P[2666]{
   GP1:
	UF : 0, UT : 6,		CONFIG : 'N U T, 0, 0, 0',
	X =  -88.796  mm,	Y =   -332.200  mm,	Z =   -251.035  mm,
	W =  90.000 deg,	P =   0.000 deg,	R =   90.000 deg
};
P[2667]{
   GP1:
	UF : 0, UT : 6,		CONFIG : 'N U T, 0, 0, 0',
	X =  -94.111  mm,	Y =   -335.387  mm,	Z =   -251.321  mm,
	W =  90.000 deg,	P =   0.000 deg,	R =   90.000 deg
};
P[2668]{
   GP1:
	UF : 0, UT : 6,		CONFIG : 'N U T, 0, 0, 0',
	X =  -94.874  mm,	Y =   -335.891  mm,	Z =   -251.475  mm,
	W =  90.000 deg,	P =   0.000 deg,	R =   90.000 deg
};
P[2669]{
   GP1:
	UF : 0, UT : 6,		CONFIG : 'N U T, 0, 0, 0',
	X =  -96.510  mm,	Y =   -336.847  mm,	Z =   -251.505  mm,
	W =  90.000 deg,	P =   0.000 deg,	R =   90.000 deg
};
P[2670]{
   GP1:
	UF : 0, UT : 6,		CONFIG : 'N U T, 0, 0, 0',
	X =  -98.758  mm,	Y =   -337.951  mm,	Z =   -251.032  mm,
	W =  90.000 deg,	P =   0.000 deg,	R =   90.000 deg
};
P[2671]{
   GP1:
	UF : 0, UT : 6,		CONFIG : 'N U T, 0, 0, 0',
	X =  -100.678  mm,	Y =   -339.223  mm,	Z =   -251.429  mm,
	W =  90.000 deg,	P =   0.000 deg,	R =   90.000 deg
};
P[2672]{
   GP1:
	UF : 0, UT : 6,		CONFIG : 'N U T, 0, 0, 0',
	X =  -102.192  mm,	Y =   -340.019  mm,	Z =   -251.240  mm,
	W =  90.000 deg,	P =   0.000 deg,	R =   90.000 deg
};
P[2673]{
   GP1:
	UF : 0, UT : 6,		CONFIG : 'N U T, 0, 0, 0',
	X =  -103.313  mm,	Y =   -340.755  mm,	Z =   -251.454  mm,
	W =  90.000 deg,	P =   0.000 deg,	R =   90.000 deg
};
P[2674]{
   GP1:
	UF : 0, UT : 6,		CONFIG : 'N U T, 0, 0, 0',
	X =  -105.295  mm,	Y =   -341.722  mm,	Z =   -251.025  mm,
	W =  90.000 deg,	P =   0.000 deg,	R =   90.000 deg
};
P[2675]{
   GP1:
	UF : 0, UT : 6,		CONFIG : 'N U T, 0, 0, 0',
	X =  -106.428  mm,	Y =   -342.386  mm,	Z =   -251.049  mm,
	W =  90.000 deg,	P =   0.000 deg,	R =   90.000 deg
};
P[2676]{
   GP1:
	UF : 0, UT : 6,		CONFIG : 'N U T, 0, 0, 0',
	X =  -108.033  mm,	Y =   -343.483  mm,	Z =   -251.461  mm,
	W =  90.000 deg,	P =   0.000 deg,	R =   90.000 deg
};
P[2677]{
   GP1:
	UF : 0, UT : 6,		CONFIG : 'N U T, 0, 0, 0',
	X =  -108.863  mm,	Y =   -343.861  mm,	Z =   -251.217  mm,
	W =  90.000 deg,	P =   0.000 deg,	R =   90.000 deg
};
P[2678]{
   GP1:
	UF : 0, UT : 6,		CONFIG : 'N U T, 0, 0, 0',
	X =  -110.601  mm,	Y =   -344.960  mm,	Z =   -251.448  mm,
	W =  90.000 deg,	P =   0.000 deg,	R =   90.000 deg
};
P[2679]{
   GP1:
	UF : 0, UT : 6,		CONFIG : 'N U T, 0, 0, 0',
	X =  -113.227  mm,	Y =   -346.434  mm,	Z =   -251.345  mm,
	W =  90.000 deg,	P =   0.000 deg,	R =   90.000 deg
};
P[2680]{
   GP1:
	UF : 0, UT : 6,		CONFIG : 'N U T, 0, 0, 0',
	X =  -116.933  mm,	Y =   -348.507  mm,	Z =   -251.183  mm,
	W =  90.000 deg,	P =   0.000 deg,	R =   90.000 deg
};
P[2681]{
   GP1:
	UF : 0, UT : 6,		CONFIG : 'N U T, 0, 0, 0',
	X =  -119.089  mm,	Y =   -350.044  mm,	Z =   -251.339  mm,
	W =  90.000 deg,	P =   0.000 deg,	R =   90.000 deg
};
P[2682]{
   GP1:
	UF : 0, UT : 6,		CONFIG : 'N U T, 0, 0, 0',
	X =  -121.292  mm,	Y =   -352.219  mm,	Z =   -251.419  mm,
	W =  90.000 deg,	P =   0.000 deg,	R =   90.000 deg
};
P[2683]{
   GP1:
	UF : 0, UT : 6,		CONFIG : 'N U T, 0, 0, 0',
	X =  -122.707  mm,	Y =   -354.283  mm,	Z =   -251.379  mm,
	W =  90.000 deg,	P =   0.000 deg,	R =   90.000 deg
};
P[2684]{
   GP1:
	UF : 0, UT : 6,		CONFIG : 'N U T, 0, 0, 0',
	X =  -123.543  mm,	Y =   -356.394  mm,	Z =   -251.512  mm,
	W =  90.000 deg,	P =   0.000 deg,	R =   90.000 deg
};
P[2685]{
   GP1:
	UF : 0, UT : 6,		CONFIG : 'N U T, 0, 0, 0',
	X =  -123.974  mm,	Y =   -357.288  mm,	Z =   -251.247  mm,
	W =  90.000 deg,	P =   0.000 deg,	R =   90.000 deg
};
P[2686]{
   GP1:
	UF : 0, UT : 6,		CONFIG : 'N U T, 0, 0, 0',
	X =  -124.171  mm,	Y =   -358.080  mm,	Z =   -251.154  mm,
	W =  90.000 deg,	P =   0.000 deg,	R =   90.000 deg
};
P[2687]{
   GP1:
	UF : 0, UT : 6,		CONFIG : 'N U T, 0, 0, 0',
	X =  -124.217  mm,	Y =   -359.462  mm,	Z =   -251.503  mm,
	W =  90.000 deg,	P =   0.000 deg,	R =   90.000 deg
};
P[2688]{
   GP1:
	UF : 0, UT : 6,		CONFIG : 'N U T, 0, 0, 0',
	X =  -124.347  mm,	Y =   -360.646  mm,	Z =   -251.277  mm,
	W =  90.000 deg,	P =   0.000 deg,	R =   90.000 deg
};
P[2689]{
   GP1:
	UF : 0, UT : 6,		CONFIG : 'N U T, 0, 0, 0',
	X =  -124.228  mm,	Y =   -361.334  mm,	Z =   -251.466  mm,
	W =  90.000 deg,	P =   0.000 deg,	R =   90.000 deg
};
P[2690]{
   GP1:
	UF : 0, UT : 6,		CONFIG : 'N U T, 0, 0, 0',
	X =  -124.026  mm,	Y =   -363.050  mm,	Z =   -251.504  mm,
	W =  90.000 deg,	P =   0.000 deg,	R =   90.000 deg
};
P[2691]{
   GP1:
	UF : 0, UT : 6,		CONFIG : 'N U T, 0, 0, 0',
	X =  -123.894  mm,	Y =   -364.249  mm,	Z =   -251.149  mm,
	W =  90.000 deg,	P =   0.000 deg,	R =   90.000 deg
};
P[2692]{
   GP1:
	UF : 0, UT : 6,		CONFIG : 'N U T, 0, 0, 0',
	X =  -123.534  mm,	Y =   -365.086  mm,	Z =   -251.490  mm,
	W =  90.000 deg,	P =   0.000 deg,	R =   90.000 deg
};
P[2693]{
   GP1:
	UF : 0, UT : 6,		CONFIG : 'N U T, 0, 0, 0',
	X =  -123.293  mm,	Y =   -365.993  mm,	Z =   -251.111  mm,
	W =  90.000 deg,	P =   0.000 deg,	R =   90.000 deg
};
P[2694]{
   GP1:
	UF : 0, UT : 6,		CONFIG : 'N U T, 0, 0, 0',
	X =  -117.435  mm,	Y =   -376.328  mm,	Z =   -251.323  mm,
	W =  90.000 deg,	P =   0.000 deg,	R =   90.000 deg
};
P[2695]{
   GP1:
	UF : 0, UT : 6,		CONFIG : 'N U T, 0, 0, 0',
	X =  -116.602  mm,	Y =   -377.647  mm,	Z =   -251.497  mm,
	W =  90.000 deg,	P =   0.000 deg,	R =   90.000 deg
};
P[2696]{
   GP1:
	UF : 0, UT : 6,		CONFIG : 'N U T, 0, 0, 0',
	X =  -116.076  mm,	Y =   -378.576  mm,	Z =   -251.473  mm,
	W =  90.000 deg,	P =   0.000 deg,	R =   90.000 deg
};
P[2697]{
   GP1:
	UF : 0, UT : 6,		CONFIG : 'N U T, 0, 0, 0',
	X =  -115.720  mm,	Y =   -379.277  mm,	Z =   -251.355  mm,
	W =  90.000 deg,	P =   0.000 deg,	R =   90.000 deg
};
P[2698]{
   GP1:
	UF : 0, UT : 6,		CONFIG : 'N U T, 0, 0, 0',
	X =  -114.684  mm,	Y =   -380.969  mm,	Z =   -251.496  mm,
	W =  90.000 deg,	P =   0.000 deg,	R =   90.000 deg
};
P[2699]{
   GP1:
	UF : 0, UT : 6,		CONFIG : 'N U T, 0, 0, 0',
	X =  -113.664  mm,	Y =   -382.827  mm,	Z =   -251.369  mm,
	W =  90.000 deg,	P =   0.000 deg,	R =   90.000 deg
};
P[2700]{
   GP1:
	UF : 0, UT : 6,		CONFIG : 'N U T, 0, 0, 0',
	X =  -112.347  mm,	Y =   -385.040  mm,	Z =   -251.463  mm,
	W =  90.000 deg,	P =   0.000 deg,	R =   90.000 deg
};
P[2701]{
   GP1:
	UF : 0, UT : 6,		CONFIG : 'N U T, 0, 0, 0',
	X =  -111.510  mm,	Y =   -386.475  mm,	Z =   -251.485  mm,
	W =  90.000 deg,	P =   0.000 deg,	R =   90.000 deg
};
P[2702]{
   GP1:
	UF : 0, UT : 6,		CONFIG : 'N U T, 0, 0, 0',
	X =  -110.653  mm,	Y =   -388.090  mm,	Z =   -251.300  mm,
	W =  90.000 deg,	P =   0.000 deg,	R =   90.000 deg
};
P[2703]{
   GP1:
	UF : 0, UT : 6,		CONFIG : 'N U T, 0, 0, 0',
	X =  -109.246  mm,	Y =   -390.539  mm,	Z =   -251.286  mm,
	W =  90.000 deg,	P =   0.000 deg,	R =   90.000 deg
};
P[2704]{
   GP1:
	UF : 0, UT : 6,		CONFIG : 'N U T, 0, 0, 0',
	X =  -107.328  mm,	Y =   -393.699  mm,	Z =   -251.513  mm,
	W =  90.000 deg,	P =   0.000 deg,	R =   90.000 deg
};
P[2705]{
   GP1:
	UF : 0, UT : 6,		CONFIG : 'N U T, 0, 0, 0',
	X =  -106.006  mm,	Y =   -396.158  mm,	Z =   -251.273  mm,
	W =  90.000 deg,	P =   0.000 deg,	R =   90.000 deg
};
P[2706]{
   GP1:
	UF : 0, UT : 6,		CONFIG : 'N U T, 0, 0, 0',
	X =  -102.398  mm,	Y =   -402.502  mm,	Z =   -251.140  mm,
	W =  90.000 deg,	P =   0.000 deg,	R =   90.000 deg
};
P[2707]{
   GP1:
	UF : 0, UT : 6,		CONFIG : 'N U T, 0, 0, 0',
	X =  -101.351  mm,	Y =   -404.270  mm,	Z =   -251.205  mm,
	W =  90.000 deg,	P =   0.000 deg,	R =   90.000 deg
};
P[2708]{
   GP1:
	UF : 0, UT : 6,		CONFIG : 'N U T, 0, 0, 0',
	X =  -100.892  mm,	Y =   -404.878  mm,	Z =   -251.465  mm,
	W =  90.000 deg,	P =   0.000 deg,	R =   90.000 deg
};
P[2709]{
   GP1:
	UF : 0, UT : 6,		CONFIG : 'N U T, 0, 0, 0',
	X =  -97.701  mm,	Y =   -410.426  mm,	Z =   -251.435  mm,
	W =  90.000 deg,	P =   0.000 deg,	R =   90.000 deg
};
P[2710]{
   GP1:
	UF : 0, UT : 6,		CONFIG : 'N U T, 0, 0, 0',
	X =  -96.296  mm,	Y =   -413.012  mm,	Z =   -251.222  mm,
	W =  90.000 deg,	P =   0.000 deg,	R =   90.000 deg
};
P[2711]{
   GP1:
	UF : 0, UT : 6,		CONFIG : 'N U T, 0, 0, 0',
	X =  -95.621  mm,	Y =   -413.979  mm,	Z =   -251.505  mm,
	W =  90.000 deg,	P =   0.000 deg,	R =   90.000 deg
};
P[2712]{
   GP1:
	UF : 0, UT : 6,		CONFIG : 'N U T, 0, 0, 0',
	X =  -94.896  mm,	Y =   -415.279  mm,	Z =   -251.445  mm,
	W =  90.000 deg,	P =   0.000 deg,	R =   90.000 deg
};
P[2713]{
   GP1:
	UF : 0, UT : 6,		CONFIG : 'N U T, 0, 0, 0',
	X =  -94.523  mm,	Y =   -416.116  mm,	Z =   -251.175  mm,
	W =  90.000 deg,	P =   0.000 deg,	R =   90.000 deg
};
P[2714]{
   GP1:
	UF : 0, UT : 6,		CONFIG : 'N U T, 0, 0, 0',
	X =  -94.072  mm,	Y =   -416.738  mm,	Z =   -251.398  mm,
	W =  90.000 deg,	P =   0.000 deg,	R =   90.000 deg
};
P[2715]{
   GP1:
	UF : 0, UT : 6,		CONFIG : 'N U T, 0, 0, 0',
	X =  -93.224  mm,	Y =   -418.286  mm,	Z =   -251.287  mm,
	W =  90.000 deg,	P =   0.000 deg,	R =   90.000 deg
};
P[2716]{
   GP1:
	UF : 0, UT : 6,		CONFIG : 'N U T, 0, 0, 0',
	X =  -92.392  mm,	Y =   -419.819  mm,	Z =   -251.157  mm,
	W =  90.000 deg,	P =   0.000 deg,	R =   90.000 deg
};
P[2717]{
   GP1:
	UF : 0, UT : 6,		CONFIG : 'N U T, 0, 0, 0',
	X =  -89.616  mm,	Y =   -424.487  mm,	Z =   -251.353  mm,
	W =  90.000 deg,	P =   0.000 deg,	R =   90.000 deg
};
P[2718]{
   GP1:
	UF : 0, UT : 6,		CONFIG : 'N U T, 0, 0, 0',
	X =  -88.935  mm,	Y =   -425.905  mm,	Z =   -251.019  mm,
	W =  90.000 deg,	P =   0.000 deg,	R =   90.000 deg
};
P[2719]{
   GP1:
	UF : 0, UT : 6,		CONFIG : 'N U T, 0, 0, 0',
	X =  -88.296  mm,	Y =   -426.877  mm,	Z =   -251.210  mm,
	W =  90.000 deg,	P =   0.000 deg,	R =   90.000 deg
};
P[2720]{
   GP1:
	UF : 0, UT : 6,		CONFIG : 'N U T, 0, 0, 0',
	X =  -87.498  mm,	Y =   -428.081  mm,	Z =   -251.458  mm,
	W =  90.000 deg,	P =   0.000 deg,	R =   90.000 deg
};
P[2721]{
   GP1:
	UF : 0, UT : 6,		CONFIG : 'N U T, 0, 0, 0',
	X =  -87.062  mm,	Y =   -428.796  mm,	Z =   -251.514  mm,
	W =  90.000 deg,	P =   0.000 deg,	R =   90.000 deg
};
P[2722]{
   GP1:
	UF : 0, UT : 6,		CONFIG : 'N U T, 0, 0, 0',
	X =  -83.860  mm,	Y =   -434.387  mm,	Z =   -251.452  mm,
	W =  90.000 deg,	P =   0.000 deg,	R =   90.000 deg
};
P[2723]{
   GP1:
	UF : 0, UT : 6,		CONFIG : 'N U T, 0, 0, 0',
	X =  -82.430  mm,	Y =   -437.003  mm,	Z =   -251.256  mm,
	W =  90.000 deg,	P =   0.000 deg,	R =   90.000 deg
};
P[2724]{
   GP1:
	UF : 0, UT : 6,		CONFIG : 'N U T, 0, 0, 0',
	X =  -80.657  mm,	Y =   -439.990  mm,	Z =   -251.371  mm,
	W =  90.000 deg,	P =   0.000 deg,	R =   90.000 deg
};
P[2725]{
   GP1:
	UF : 0, UT : 6,		CONFIG : 'N U T, 0, 0, 0',
	X =  -80.143  mm,	Y =   -440.820  mm,	Z =   -251.456  mm,
	W =  90.000 deg,	P =   0.000 deg,	R =   90.000 deg
};
P[2726]{
   GP1:
	UF : 0, UT : 6,		CONFIG : 'N U T, 0, 0, 0',
	X =  -79.054  mm,	Y =   -442.851  mm,	Z =   -251.254  mm,
	W =  90.000 deg,	P =   0.000 deg,	R =   90.000 deg
};
P[2727]{
   GP1:
	UF : 0, UT : 6,		CONFIG : 'N U T, 0, 0, 0',
	X =  -77.555  mm,	Y =   -445.264  mm,	Z =   -251.509  mm,
	W =  90.000 deg,	P =   0.000 deg,	R =   90.000 deg
};
P[2728]{
   GP1:
	UF : 0, UT : 6,		CONFIG : 'N U T, 0, 0, 0',
	X =  -75.494  mm,	Y =   -449.012  mm,	Z =   -251.260  mm,
	W =  90.000 deg,	P =   0.000 deg,	R =   90.000 deg
};
P[2729]{
   GP1:
	UF : 0, UT : 6,		CONFIG : 'N U T, 0, 0, 0',
	X =  -74.771  mm,	Y =   -450.179  mm,	Z =   -251.380  mm,
	W =  90.000 deg,	P =   0.000 deg,	R =   90.000 deg
};
P[2730]{
   GP1:
	UF : 0, UT : 6,		CONFIG : 'N U T, 0, 0, 0',
	X =  -73.079  mm,	Y =   -453.059  mm,	Z =   -251.451  mm,
	W =  90.000 deg,	P =   0.000 deg,	R =   90.000 deg
};
P[2731]{
   GP1:
	UF : 0, UT : 6,		CONFIG : 'N U T, 0, 0, 0',
	X =  -68.696  mm,	Y =   -460.609  mm,	Z =   -251.506  mm,
	W =  90.000 deg,	P =   0.000 deg,	R =   90.000 deg
};
P[2732]{
   GP1:
	UF : 0, UT : 6,		CONFIG : 'N U T, 0, 0, 0',
	X =  -68.326  mm,	Y =   -461.356  mm,	Z =   -251.359  mm,
	W =  90.000 deg,	P =   0.000 deg,	R =   90.000 deg
};
P[2733]{
   GP1:
	UF : 0, UT : 6,		CONFIG : 'N U T, 0, 0, 0',
	X =  -67.778  mm,	Y =   -462.396  mm,	Z =   -251.232  mm,
	W =  90.000 deg,	P =   0.000 deg,	R =   90.000 deg
};
P[2734]{
   GP1:
	UF : 0, UT : 6,		CONFIG : 'N U T, 0, 0, 0',
	X =  -67.192  mm,	Y =   -463.250  mm,	Z =   -251.458  mm,
	W =  90.000 deg,	P =   0.000 deg,	R =   90.000 deg
};
P[2735]{
   GP1:
	UF : 0, UT : 6,		CONFIG : 'N U T, 0, 0, 0',
	X =  -64.146  mm,	Y =   -468.762  mm,	Z =   -251.125  mm,
	W =  90.000 deg,	P =   0.000 deg,	R =   90.000 deg
};
P[2736]{
   GP1:
	UF : 0, UT : 6,		CONFIG : 'N U T, 0, 0, 0',
	X =  -62.301  mm,	Y =   -471.708  mm,	Z =   -251.474  mm,
	W =  90.000 deg,	P =   0.000 deg,	R =   90.000 deg
};
P[2737]{
   GP1:
	UF : 0, UT : 6,		CONFIG : 'N U T, 0, 0, 0',
	X =  -60.967  mm,	Y =   -474.301  mm,	Z =   -251.079  mm,
	W =  90.000 deg,	P =   0.000 deg,	R =   90.000 deg
};
P[2738]{
   GP1:
	UF : 0, UT : 6,		CONFIG : 'N U T, 0, 0, 0',
	X =  -59.945  mm,	Y =   -475.996  mm,	Z =   -251.183  mm,
	W =  90.000 deg,	P =   0.000 deg,	R =   90.000 deg
};
P[2739]{
   GP1:
	UF : 0, UT : 6,		CONFIG : 'N U T, 0, 0, 0',
	X =  -56.961  mm,	Y =   -481.089  mm,	Z =   -251.291  mm,
	W =  90.000 deg,	P =   0.000 deg,	R =   90.000 deg
};
P[2740]{
   GP1:
	UF : 0, UT : 6,		CONFIG : 'N U T, 0, 0, 0',
	X =  -55.926  mm,	Y =   -482.733  mm,	Z =   -251.499  mm,
	W =  90.000 deg,	P =   0.000 deg,	R =   90.000 deg
};
P[2741]{
   GP1:
	UF : 0, UT : 6,		CONFIG : 'N U T, 0, 0, 0',
	X =  -55.119  mm,	Y =   -484.466  mm,	Z =   -251.027  mm,
	W =  90.000 deg,	P =   0.000 deg,	R =   90.000 deg
};
P[2742]{
   GP1:
	UF : 0, UT : 6,		CONFIG : 'N U T, 0, 0, 0',
	X =  -52.807  mm,	Y =   -488.183  mm,	Z =   -251.430  mm,
	W =  90.000 deg,	P =   0.000 deg,	R =   90.000 deg
};
P[2743]{
   GP1:
	UF : 0, UT : 6,		CONFIG : 'N U T, 0, 0, 0',
	X =  -52.049  mm,	Y =   -489.711  mm,	Z =   -251.128  mm,
	W =  90.000 deg,	P =   0.000 deg,	R =   90.000 deg
};
P[2744]{
   GP1:
	UF : 0, UT : 6,		CONFIG : 'N U T, 0, 0, 0',
	X =  -48.701  mm,	Y =   -495.270  mm,	Z =   -251.462  mm,
	W =  90.000 deg,	P =   0.000 deg,	R =   90.000 deg
};
P[2745]{
   GP1:
	UF : 0, UT : 6,		CONFIG : 'N U T, 0, 0, 0',
	X =  -48.119  mm,	Y =   -496.321  mm,	Z =   -251.403  mm,
	W =  90.000 deg,	P =   0.000 deg,	R =   90.000 deg
};
P[2746]{
   GP1:
	UF : 0, UT : 6,		CONFIG : 'N U T, 0, 0, 0',
	X =  -46.469  mm,	Y =   -499.194  mm,	Z =   -251.385  mm,
	W =  90.000 deg,	P =   0.000 deg,	R =   90.000 deg
};
P[2747]{
   GP1:
	UF : 0, UT : 6,		CONFIG : 'N U T, 0, 0, 0',
	X =  -46.266  mm,	Y =   -499.788  mm,	Z =   -251.042  mm,
	W =  90.000 deg,	P =   0.000 deg,	R =   90.000 deg
};
P[2748]{
   GP1:
	UF : 0, UT : 6,		CONFIG : 'N U T, 0, 0, 0',
	X =  -45.082  mm,	Y =   -501.624  mm,	Z =   -251.345  mm,
	W =  90.000 deg,	P =   0.000 deg,	R =   90.000 deg
};
P[2749]{
   GP1:
	UF : 0, UT : 6,		CONFIG : 'N U T, 0, 0, 0',
	X =  -44.497  mm,	Y =   -502.677  mm,	Z =   -251.288  mm,
	W =  90.000 deg,	P =   0.000 deg,	R =   90.000 deg
};
P[2750]{
   GP1:
	UF : 0, UT : 6,		CONFIG : 'N U T, 0, 0, 0',
	X =  -44.054  mm,	Y =   -503.435  mm,	Z =   -251.301  mm,
	W =  90.000 deg,	P =   0.000 deg,	R =   90.000 deg
};
P[2751]{
   GP1:
	UF : 0, UT : 6,		CONFIG : 'N U T, 0, 0, 0',
	X =  -41.974  mm,	Y =   -507.109  mm,	Z =   -251.201  mm,
	W =  90.000 deg,	P =   0.000 deg,	R =   90.000 deg
};
P[2752]{
   GP1:
	UF : 0, UT : 6,		CONFIG : 'N U T, 0, 0, 0',
	X =  -41.447  mm,	Y =   -507.963  mm,	Z =   -251.281  mm,
	W =  90.000 deg,	P =   0.000 deg,	R =   90.000 deg
};
P[2753]{
   GP1:
	UF : 0, UT : 6,		CONFIG : 'N U T, 0, 0, 0',
	X =  -40.849  mm,	Y =   -508.939  mm,	Z =   -251.367  mm,
	W =  90.000 deg,	P =   0.000 deg,	R =   90.000 deg
};
P[2754]{
   GP1:
	UF : 0, UT : 6,		CONFIG : 'N U T, 0, 0, 0',
	X =  -39.722  mm,	Y =   -510.925  mm,	Z =   -251.316  mm,
	W =  90.000 deg,	P =   0.000 deg,	R =   90.000 deg
};
P[2755]{
   GP1:
	UF : 0, UT : 6,		CONFIG : 'N U T, 0, 0, 0',
	X =  -38.820  mm,	Y =   -512.403  mm,	Z =   -251.437  mm,
	W =  90.000 deg,	P =   0.000 deg,	R =   90.000 deg
};
P[2756]{
   GP1:
	UF : 0, UT : 6,		CONFIG : 'N U T, 0, 0, 0',
	X =  -36.903  mm,	Y =   -515.957  mm,	Z =   -251.109  mm,
	W =  90.000 deg,	P =   0.000 deg,	R =   90.000 deg
};
P[2757]{
   GP1:
	UF : 0, UT : 6,		CONFIG : 'N U T, 0, 0, 0',
	X =  -35.467  mm,	Y =   -518.413  mm,	Z =   -251.152  mm,
	W =  90.000 deg,	P =   0.000 deg,	R =   90.000 deg
};
P[2758]{
   GP1:
	UF : 0, UT : 6,		CONFIG : 'N U T, 0, 0, 0',
	X =  -34.404  mm,	Y =   -520.025  mm,	Z =   -251.475  mm,
	W =  90.000 deg,	P =   0.000 deg,	R =   90.000 deg
};
P[2759]{
   GP1:
	UF : 0, UT : 6,		CONFIG : 'N U T, 0, 0, 0',
	X =  -32.513  mm,	Y =   -523.279  mm,	Z =   -251.503  mm,
	W =  90.000 deg,	P =   0.000 deg,	R =   90.000 deg
};
P[2760]{
   GP1:
	UF : 0, UT : 6,		CONFIG : 'N U T, 0, 0, 0',
	X =  -32.011  mm,	Y =   -524.184  mm,	Z =   -251.452  mm,
	W =  90.000 deg,	P =   0.000 deg,	R =   90.000 deg
};
P[2761]{
   GP1:
	UF : 0, UT : 6,		CONFIG : 'N U T, 0, 0, 0',
	X =  -30.707  mm,	Y =   -526.524  mm,	Z =   -251.340  mm,
	W =  90.000 deg,	P =   0.000 deg,	R =   90.000 deg
};
P[2762]{
   GP1:
	UF : 0, UT : 6,		CONFIG : 'N U T, 0, 0, 0',
	X =  -29.786  mm,	Y =   -528.328  mm,	Z =   -251.045  mm,
	W =  90.000 deg,	P =   0.000 deg,	R =   90.000 deg
};
P[2763]{
   GP1:
	UF : 0, UT : 6,		CONFIG : 'N U T, 0, 0, 0',
	X =  -28.612  mm,	Y =   -530.119  mm,	Z =   -251.386  mm,
	W =  90.000 deg,	P =   0.000 deg,	R =   90.000 deg
};
P[2764]{
   GP1:
	UF : 0, UT : 6,		CONFIG : 'N U T, 0, 0, 0',
	X =  -28.076  mm,	Y =   -530.989  mm,	Z =   -251.466  mm,
	W =  90.000 deg,	P =   0.000 deg,	R =   90.000 deg
};
P[2765]{
   GP1:
	UF : 0, UT : 6,		CONFIG : 'N U T, 0, 0, 0',
	X =  -25.936  mm,	Y =   -534.844  mm,	Z =   -251.260  mm,
	W =  90.000 deg,	P =   0.000 deg,	R =   90.000 deg
};
P[2766]{
   GP1:
	UF : 0, UT : 6,		CONFIG : 'N U T, 0, 0, 0',
	X =  -25.504  mm,	Y =   -535.459  mm,	Z =   -251.446  mm,
	W =  90.000 deg,	P =   0.000 deg,	R =   90.000 deg
};
P[2767]{
   GP1:
	UF : 0, UT : 6,		CONFIG : 'N U T, 0, 0, 0',
	X =  -24.086  mm,	Y =   -537.957  mm,	Z =   -251.386  mm,
	W =  90.000 deg,	P =   0.000 deg,	R =   90.000 deg
};
P[2768]{
   GP1:
	UF : 0, UT : 6,		CONFIG : 'N U T, 0, 0, 0',
	X =  -21.165  mm,	Y =   -542.983  mm,	Z =   -251.433  mm,
	W =  90.000 deg,	P =   0.000 deg,	R =   90.000 deg
};
P[2769]{
   GP1:
	UF : 0, UT : 6,		CONFIG : 'N U T, 0, 0, 0',
	X =  -20.589  mm,	Y =   -543.926  mm,	Z =   -251.508  mm,
	W =  90.000 deg,	P =   0.000 deg,	R =   90.000 deg
};
P[2770]{
   GP1:
	UF : 0, UT : 6,		CONFIG : 'N U T, 0, 0, 0',
	X =  -15.957  mm,	Y =   -552.282  mm,	Z =   -251.040  mm,
	W =  90.000 deg,	P =   0.000 deg,	R =   90.000 deg
};
P[2771]{
   GP1:
	UF : 0, UT : 6,		CONFIG : 'N U T, 0, 0, 0',
	X =  -14.354  mm,	Y =   -554.787  mm,	Z =   -251.423  mm,
	W =  90.000 deg,	P =   0.000 deg,	R =   90.000 deg
};
P[2772]{
   GP1:
	UF : 0, UT : 6,		CONFIG : 'N U T, 0, 0, 0',
	X =  -11.877  mm,	Y =   -559.032  mm,	Z =   -251.483  mm,
	W =  90.000 deg,	P =   0.000 deg,	R =   90.000 deg
};
P[2773]{
   GP1:
	UF : 0, UT : 6,		CONFIG : 'N U T, 0, 0, 0',
	X =  -8.884  mm,	Y =   -564.221  mm,	Z =   -251.478  mm,
	W =  90.000 deg,	P =   0.000 deg,	R =   90.000 deg
};
P[2774]{
   GP1:
	UF : 0, UT : 6,		CONFIG : 'N U T, 0, 0, 0',
	X =  -7.979  mm,	Y =   -565.863  mm,	Z =   -251.375  mm,
	W =  90.000 deg,	P =   0.000 deg,	R =   90.000 deg
};
P[2775]{
   GP1:
	UF : 0, UT : 6,		CONFIG : 'N U T, 0, 0, 0',
	X =  -7.245  mm,	Y =   -567.071  mm,	Z =   -251.459  mm,
	W =  90.000 deg,	P =   0.000 deg,	R =   90.000 deg
};
P[2776]{
   GP1:
	UF : 0, UT : 6,		CONFIG : 'N U T, 0, 0, 0',
	X =  -6.779  mm,	Y =   -567.853  mm,	Z =   -251.496  mm,
	W =  90.000 deg,	P =   0.000 deg,	R =   90.000 deg
};
P[2777]{
   GP1:
	UF : 0, UT : 6,		CONFIG : 'N U T, 0, 0, 0',
	X =  -5.072  mm,	Y =   -570.860  mm,	Z =   -251.425  mm,
	W =  90.000 deg,	P =   0.000 deg,	R =   90.000 deg
};
P[2778]{
   GP1:
	UF : 0, UT : 6,		CONFIG : 'N U T, 0, 0, 0',
	X =  -2.813  mm,	Y =   -574.858  mm,	Z =   -251.308  mm,
	W =  90.000 deg,	P =   0.000 deg,	R =   90.000 deg
};
P[2779]{
   GP1:
	UF : 0, UT : 6,		CONFIG : 'N U T, 0, 0, 0',
	X =  -1.783  mm,	Y =   -576.767  mm,	Z =   -251.131  mm,
	W =  90.000 deg,	P =   0.000 deg,	R =   90.000 deg
};
P[2780]{
   GP1:
	UF : 0, UT : 6,		CONFIG : 'N U T, 0, 0, 0',
	X =  -1.133  mm,	Y =   -577.837  mm,	Z =   -251.208  mm,
	W =  90.000 deg,	P =   0.000 deg,	R =   90.000 deg
};
P[2781]{
   GP1:
	UF : 0, UT : 6,		CONFIG : 'N U T, 0, 0, 0',
	X =  -0.576  mm,	Y =   -578.717  mm,	Z =   -251.326  mm,
	W =  90.000 deg,	P =   0.000 deg,	R =   90.000 deg
};
P[2782]{
   GP1:
	UF : 0, UT : 6,		CONFIG : 'N U T, 0, 0, 0',
	X =  1.420  mm,	Y =   -582.138  mm,	Z =   -251.378  mm,
	W =  90.000 deg,	P =   0.000 deg,	R =   90.000 deg
};
P[2783]{
   GP1:
	UF : 0, UT : 6,		CONFIG : 'N U T, 0, 0, 0',
	X =  2.275  mm,	Y =   -583.540  mm,	Z =   -251.487  mm,
	W =  90.000 deg,	P =   0.000 deg,	R =   90.000 deg
};
P[2784]{
   GP1:
	UF : 0, UT : 6,		CONFIG : 'N U T, 0, 0, 0',
	X =  2.580  mm,	Y =   -584.263  mm,	Z =   -251.216  mm,
	W =  90.000 deg,	P =   0.000 deg,	R =   90.000 deg
};
P[2785]{
   GP1:
	UF : 0, UT : 6,		CONFIG : 'N U T, 0, 0, 0',
	X =  3.375  mm,	Y =   -585.474  mm,	Z =   -251.448  mm,
	W =  90.000 deg,	P =   0.000 deg,	R =   90.000 deg
};
P[2786]{
   GP1:
	UF : 0, UT : 6,		CONFIG : 'N U T, 0, 0, 0',
	X =  6.611  mm,	Y =   -591.060  mm,	Z =   -251.474  mm,
	W =  90.000 deg,	P =   0.000 deg,	R =   90.000 deg
};
P[2787]{
   GP1:
	UF : 0, UT : 6,		CONFIG : 'N U T, 0, 0, 0',
	X =  8.109  mm,	Y =   -593.784  mm,	Z =   -251.289  mm,
	W =  90.000 deg,	P =   0.000 deg,	R =   90.000 deg
};
P[2788]{
   GP1:
	UF : 0, UT : 6,		CONFIG : 'N U T, 0, 0, 0',
	X =  8.696  mm,	Y =   -594.768  mm,	Z =   -251.336  mm,
	W =  90.000 deg,	P =   0.000 deg,	R =   90.000 deg
};
P[2789]{
   GP1:
	UF : 0, UT : 6,		CONFIG : 'N U T, 0, 0, 0',
	X =  9.244  mm,	Y =   -595.621  mm,	Z =   -251.473  mm,
	W =  90.000 deg,	P =   0.000 deg,	R =   90.000 deg
};
P[2790]{
   GP1:
	UF : 0, UT : 6,		CONFIG : 'N U T, 0, 0, 0',
	X =  11.919  mm,	Y =   -600.232  mm,	Z =   -251.502  mm,
	W =  90.000 deg,	P =   0.000 deg,	R =   90.000 deg
};
P[2791]{
   GP1:
	UF : 0, UT : 6,		CONFIG : 'N U T, 0, 0, 0',
	X =  12.721  mm,	Y =   -601.663  mm,	Z =   -251.443  mm,
	W =  90.000 deg,	P =   0.000 deg,	R =   90.000 deg
};
P[2792]{
   GP1:
	UF : 0, UT : 6,		CONFIG : 'N U T, 0, 0, 0',
	X =  14.239  mm,	Y =   -604.336  mm,	Z =   -251.383  mm,
	W =  90.000 deg,	P =   0.000 deg,	R =   90.000 deg
};
P[2793]{
   GP1:
	UF : 0, UT : 6,		CONFIG : 'N U T, 0, 0, 0',
	X =  15.858  mm,	Y =   -607.148  mm,	Z =   -251.369  mm,
	W =  90.000 deg,	P =   0.000 deg,	R =   90.000 deg
};
P[2794]{
   GP1:
	UF : 0, UT : 6,		CONFIG : 'N U T, 0, 0, 0',
	X =  16.759  mm,	Y =   -608.769  mm,	Z =   -251.287  mm,
	W =  90.000 deg,	P =   0.000 deg,	R =   90.000 deg
};
P[2795]{
   GP1:
	UF : 0, UT : 6,		CONFIG : 'N U T, 0, 0, 0',
	X =  18.576  mm,	Y =   -611.947  mm,	Z =   -251.243  mm,
	W =  90.000 deg,	P =   0.000 deg,	R =   90.000 deg
};
P[2796]{
   GP1:
	UF : 0, UT : 6,		CONFIG : 'N U T, 0, 0, 0',
	X =  19.161  mm,	Y =   -612.944  mm,	Z =   -251.266  mm,
	W =  90.000 deg,	P =   0.000 deg,	R =   90.000 deg
};
P[2797]{
   GP1:
	UF : 0, UT : 6,		CONFIG : 'N U T, 0, 0, 0',
	X =  19.658  mm,	Y =   -613.779  mm,	Z =   -251.302  mm,
	W =  90.000 deg,	P =   0.000 deg,	R =   90.000 deg
};
P[2798]{
   GP1:
	UF : 0, UT : 6,		CONFIG : 'N U T, 0, 0, 0',
	X =  20.200  mm,	Y =   -614.689  mm,	Z =   -251.343  mm,
	W =  90.000 deg,	P =   0.000 deg,	R =   90.000 deg
};
P[2799]{
   GP1:
	UF : 0, UT : 6,		CONFIG : 'N U T, 0, 0, 0',
	X =  20.838  mm,	Y =   -615.769  mm,	Z =   -251.379  mm,
	W =  90.000 deg,	P =   0.000 deg,	R =   90.000 deg
};
P[2800]{
   GP1:
	UF : 0, UT : 6,		CONFIG : 'N U T, 0, 0, 0',
	X =  24.409  mm,	Y =   -621.940  mm,	Z =   -251.398  mm,
	W =  90.000 deg,	P =   0.000 deg,	R =   90.000 deg
};
P[2801]{
   GP1:
	UF : 0, UT : 6,		CONFIG : 'N U T, 0, 0, 0',
	X =  26.270  mm,	Y =   -625.160  mm,	Z =   -251.402  mm,
	W =  90.000 deg,	P =   0.000 deg,	R =   90.000 deg
};
P[2802]{
   GP1:
	UF : 0, UT : 6,		CONFIG : 'N U T, 0, 0, 0',
	X =  27.634  mm,	Y =   -627.517  mm,	Z =   -251.408  mm,
	W =  90.000 deg,	P =   0.000 deg,	R =   90.000 deg
};
P[2803]{
   GP1:
	UF : 0, UT : 6,		CONFIG : 'N U T, 0, 0, 0',
	X =  28.698  mm,	Y =   -629.325  mm,	Z =   -251.457  mm,
	W =  90.000 deg,	P =   0.000 deg,	R =   90.000 deg
};
P[2804]{
   GP1:
	UF : 0, UT : 6,		CONFIG : 'N U T, 0, 0, 0',
	X =  29.024  mm,	Y =   -630.020  mm,	Z =   -251.275  mm,
	W =  90.000 deg,	P =   0.000 deg,	R =   90.000 deg
};
P[2805]{
   GP1:
	UF : 0, UT : 6,		CONFIG : 'N U T, 0, 0, 0',
	X =  30.603  mm,	Y =   -632.779  mm,	Z =   -251.241  mm,
	W =  90.000 deg,	P =   0.000 deg,	R =   90.000 deg
};
P[2806]{
   GP1:
	UF : 0, UT : 6,		CONFIG : 'N U T, 0, 0, 0',
	X =  31.111  mm,	Y =   -633.721  mm,	Z =   -251.153  mm,
	W =  90.000 deg,	P =   0.000 deg,	R =   90.000 deg
};
P[2807]{
   GP1:
	UF : 0, UT : 6,		CONFIG : 'N U T, 0, 0, 0',
	X =  31.623  mm,	Y =   -634.667  mm,	Z =   -251.072  mm,
	W =  90.000 deg,	P =   0.000 deg,	R =   90.000 deg
};
P[2808]{
   GP1:
	UF : 0, UT : 6,		CONFIG : 'N U T, 0, 0, 0',
	X =  33.028  mm,	Y =   -637.101  mm,	Z =   -251.068  mm,
	W =  90.000 deg,	P =   0.000 deg,	R =   90.000 deg
};
P[2809]{
   GP1:
	UF : 0, UT : 6,		CONFIG : 'N U T, 0, 0, 0',
	X =  33.530  mm,	Y =   -637.742  mm,	Z =   -251.391  mm,
	W =  90.000 deg,	P =   0.000 deg,	R =   90.000 deg
};
P[2810]{
   GP1:
	UF : 0, UT : 6,		CONFIG : 'N U T, 0, 0, 0',
	X =  35.590  mm,	Y =   -641.325  mm,	Z =   -251.365  mm,
	W =  90.000 deg,	P =   0.000 deg,	R =   90.000 deg
};
P[2811]{
   GP1:
	UF : 0, UT : 6,		CONFIG : 'N U T, 0, 0, 0',
	X =  37.083  mm,	Y =   -644.038  mm,	Z =   -251.189  mm,
	W =  90.000 deg,	P =   0.000 deg,	R =   90.000 deg
};
P[2812]{
   GP1:
	UF : 0, UT : 6,		CONFIG : 'N U T, 0, 0, 0',
	X =  38.478  mm,	Y =   -646.252  mm,	Z =   -251.473  mm,
	W =  90.000 deg,	P =   0.000 deg,	R =   90.000 deg
};
P[2813]{
   GP1:
	UF : 0, UT : 6,		CONFIG : 'N U T, 0, 0, 0',
	X =  39.055  mm,	Y =   -647.577  mm,	Z =   -251.016  mm,
	W =  90.000 deg,	P =   0.000 deg,	R =   90.000 deg
};
P[2814]{
   GP1:
	UF : 0, UT : 6,		CONFIG : 'N U T, 0, 0, 0',
	X =  42.203  mm,	Y =   -652.875  mm,	Z =   -251.234  mm,
	W =  90.000 deg,	P =   0.000 deg,	R =   90.000 deg
};
P[2815]{
   GP1:
	UF : 0, UT : 6,		CONFIG : 'N U T, 0, 0, 0',
	X =  42.873  mm,	Y =   -653.847  mm,	Z =   -251.496  mm,
	W =  90.000 deg,	P =   0.000 deg,	R =   90.000 deg
};
P[2816]{
   GP1:
	UF : 0, UT : 6,		CONFIG : 'N U T, 0, 0, 0',
	X =  43.459  mm,	Y =   -654.879  mm,	Z =   -251.471  mm,
	W =  90.000 deg,	P =   0.000 deg,	R =   90.000 deg
};
P[2817]{
   GP1:
	UF : 0, UT : 6,		CONFIG : 'N U T, 0, 0, 0',
	X =  44.323  mm,	Y =   -656.489  mm,	Z =   -251.312  mm,
	W =  90.000 deg,	P =   0.000 deg,	R =   90.000 deg
};
P[2818]{
   GP1:
	UF : 0, UT : 6,		CONFIG : 'N U T, 0, 0, 0',
	X =  45.796  mm,	Y =   -659.114  mm,	Z =   -251.209  mm,
	W =  90.000 deg,	P =   0.000 deg,	R =   90.000 deg
};
P[2819]{
   GP1:
	UF : 0, UT : 6,		CONFIG : 'N U T, 0, 0, 0',
	X =  47.101  mm,	Y =   -661.258  mm,	Z =   -251.372  mm,
	W =  90.000 deg,	P =   0.000 deg,	R =   90.000 deg
};
P[2820]{
   GP1:
	UF : 0, UT : 6,		CONFIG : 'N U T, 0, 0, 0',
	X =  49.273  mm,	Y =   -664.958  mm,	Z =   -251.458  mm,
	W =  90.000 deg,	P =   0.000 deg,	R =   90.000 deg
};
P[2821]{
   GP1:
	UF : 0, UT : 6,		CONFIG : 'N U T, 0, 0, 0',
	X =  50.034  mm,	Y =   -666.310  mm,	Z =   -251.409  mm,
	W =  90.000 deg,	P =   0.000 deg,	R =   90.000 deg
};
P[2822]{
   GP1:
	UF : 0, UT : 6,		CONFIG : 'N U T, 0, 0, 0',
	X =  50.645  mm,	Y =   -667.304  mm,	Z =   -251.268  mm,
	W =  90.000 deg,	P =   0.000 deg,	R =   90.000 deg
};
P[2823]{
   GP1:
	UF : 0, UT : 6,		CONFIG : 'N U T, 0, 0, 0',
	X =  51.316  mm,	Y =   -668.207  mm,	Z =   -251.328  mm,
	W =  90.000 deg,	P =   0.000 deg,	R =   90.000 deg
};
P[2824]{
   GP1:
	UF : 0, UT : 6,		CONFIG : 'N U T, 0, 0, 0',
	X =  52.230  mm,	Y =   -669.410  mm,	Z =   -251.133  mm,
	W =  90.000 deg,	P =   0.000 deg,	R =   90.000 deg
};
P[2825]{
   GP1:
	UF : 0, UT : 6,		CONFIG : 'N U T, 0, 0, 0',
	X =  53.416  mm,	Y =   -670.323  mm,	Z =   -251.491  mm,
	W =  90.000 deg,	P =   0.000 deg,	R =   90.000 deg
};
P[2826]{
   GP1:
	UF : 0, UT : 6,		CONFIG : 'N U T, 0, 0, 0',
	X =  54.372  mm,	Y =   -671.033  mm,	Z =   -251.512  mm,
	W =  90.000 deg,	P =   0.000 deg,	R =   90.000 deg
};
P[2827]{
   GP1:
	UF : 0, UT : 6,		CONFIG : 'N U T, 0, 0, 0',
	X =  55.316  mm,	Y =   -671.802  mm,	Z =   -251.215  mm,
	W =  90.000 deg,	P =   0.000 deg,	R =   90.000 deg
};
P[2828]{
   GP1:
	UF : 0, UT : 6,		CONFIG : 'N U T, 0, 0, 0',
	X =  60.468  mm,	Y =   -673.560  mm,	Z =   -251.089  mm,
	W =  90.000 deg,	P =   0.000 deg,	R =   90.000 deg
};
P[2829]{
   GP1:
	UF : 0, UT : 6,		CONFIG : 'N U T, 0, 0, 0',
	X =  61.166  mm,	Y =   -673.584  mm,	Z =   -251.188  mm,
	W =  90.000 deg,	P =   0.000 deg,	R =   90.000 deg
};
P[2830]{
   GP1:
	UF : 0, UT : 6,		CONFIG : 'N U T, 0, 0, 0',
	X =  62.620  mm,	Y =   -673.412  mm,	Z =   -251.473  mm,
	W =  90.000 deg,	P =   0.000 deg,	R =   90.000 deg
};
P[2831]{
   GP1:
	UF : 0, UT : 6,		CONFIG : 'N U T, 0, 0, 0',
	X =  63.514  mm,	Y =   -673.561  mm,	Z =   -251.085  mm,
	W =  90.000 deg,	P =   0.000 deg,	R =   90.000 deg
};
P[2832]{
   GP1:
	UF : 0, UT : 6,		CONFIG : 'N U T, 0, 0, 0',
	X =  64.691  mm,	Y =   -673.218  mm,	Z =   -251.321  mm,
	W =  90.000 deg,	P =   0.000 deg,	R =   90.000 deg
};
P[2833]{
   GP1:
	UF : 0, UT : 6,		CONFIG : 'N U T, 0, 0, 0',
	X =  67.176  mm,	Y =   -672.394  mm,	Z =   -251.458  mm,
	W =  90.000 deg,	P =   0.000 deg,	R =   90.000 deg
};
P[2834]{
   GP1:
	UF : 0, UT : 6,		CONFIG : 'N U T, 0, 0, 0',
	X =  71.284  mm,	Y =   -670.282  mm,	Z =   -251.360  mm,
	W =  90.000 deg,	P =   0.000 deg,	R =   90.000 deg
};
P[2835]{
   GP1:
	UF : 0, UT : 6,		CONFIG : 'N U T, 0, 0, 0',
	X =  74.075  mm,	Y =   -668.766  mm,	Z =   -251.129  mm,
	W =  90.000 deg,	P =   0.000 deg,	R =   90.000 deg
};
P[2836]{
   GP1:
	UF : 0, UT : 6,		CONFIG : 'N U T, 0, 0, 0',
	X =  74.898  mm,	Y =   -668.189  mm,	Z =   -251.376  mm,
	W =  90.000 deg,	P =   0.000 deg,	R =   90.000 deg
};
P[2837]{
   GP1:
	UF : 0, UT : 6,		CONFIG : 'N U T, 0, 0, 0',
	X =  76.634  mm,	Y =   -667.160  mm,	Z =   -251.438  mm,
	W =  90.000 deg,	P =   0.000 deg,	R =   90.000 deg
};
P[2838]{
   GP1:
	UF : 0, UT : 6,		CONFIG : 'N U T, 0, 0, 0',
	X =  78.182  mm,	Y =   -666.329  mm,	Z =   -251.288  mm,
	W =  90.000 deg,	P =   0.000 deg,	R =   90.000 deg
};
P[2839]{
   GP1:
	UF : 0, UT : 6,		CONFIG : 'N U T, 0, 0, 0',
	X =  81.400  mm,	Y =   -664.411  mm,	Z =   -251.431  mm,
	W =  90.000 deg,	P =   0.000 deg,	R =   90.000 deg
};
P[2840]{
   GP1:
	UF : 0, UT : 6,		CONFIG : 'N U T, 0, 0, 0',
	X =  83.844  mm,	Y =   -663.171  mm,	Z =   -251.017  mm,
	W =  90.000 deg,	P =   0.000 deg,	R =   90.000 deg
};
P[2841]{
   GP1:
	UF : 0, UT : 6,		CONFIG : 'N U T, 0, 0, 0',
	X =  84.752  mm,	Y =   -662.447  mm,	Z =   -251.500  mm,
	W =  90.000 deg,	P =   0.000 deg,	R =   90.000 deg
};
P[2842]{
   GP1:
	UF : 0, UT : 6,		CONFIG : 'N U T, 0, 0, 0',
	X =  86.033  mm,	Y =   -661.871  mm,	Z =   -251.105  mm,
	W =  90.000 deg,	P =   0.000 deg,	R =   90.000 deg
};
P[2843]{
   GP1:
	UF : 0, UT : 6,		CONFIG : 'N U T, 0, 0, 0',
	X =  94.303  mm,	Y =   -657.067  mm,	Z =   -251.174  mm,
	W =  90.000 deg,	P =   0.000 deg,	R =   90.000 deg
};
P[2844]{
   GP1:
	UF : 0, UT : 6,		CONFIG : 'N U T, 0, 0, 0',
	X =  95.219  mm,	Y =   -656.581  mm,	Z =   -251.072  mm,
	W =  90.000 deg,	P =   0.000 deg,	R =   90.000 deg
};
P[2845]{
   GP1:
	UF : 0, UT : 6,		CONFIG : 'N U T, 0, 0, 0',
	X =  97.107  mm,	Y =   -655.492  mm,	Z =   -251.067  mm,
	W =  90.000 deg,	P =   0.000 deg,	R =   90.000 deg
};
P[2846]{
   GP1:
	UF : 0, UT : 6,		CONFIG : 'N U T, 0, 0, 0',
	X =  97.790  mm,	Y =   -654.951  mm,	Z =   -251.423  mm,
	W =  90.000 deg,	P =   0.000 deg,	R =   90.000 deg
};
P[2847]{
   GP1:
	UF : 0, UT : 6,		CONFIG : 'N U T, 0, 0, 0',
	X =  99.311  mm,	Y =   -654.078  mm,	Z =   -251.410  mm,
	W =  90.000 deg,	P =   0.000 deg,	R =   90.000 deg
};
P[2848]{
   GP1:
	UF : 0, UT : 6,		CONFIG : 'N U T, 0, 0, 0',
	X =  102.841  mm,	Y =   -652.160  mm,	Z =   -251.120  mm,
	W =  90.000 deg,	P =   0.000 deg,	R =   90.000 deg
};
P[2849]{
   GP1:
	UF : 0, UT : 6,		CONFIG : 'N U T, 0, 0, 0',
	X =  105.417  mm,	Y =   -650.662  mm,	Z =   -251.144  mm,
	W =  90.000 deg,	P =   0.000 deg,	R =   90.000 deg
};
P[2850]{
   GP1:
	UF : 0, UT : 6,		CONFIG : 'N U T, 0, 0, 0',
	X =  107.018  mm,	Y =   -649.683  mm,	Z =   -251.277  mm,
	W =  90.000 deg,	P =   0.000 deg,	R =   90.000 deg
};
P[2851]{
   GP1:
	UF : 0, UT : 6,		CONFIG : 'N U T, 0, 0, 0',
	X =  110.149  mm,	Y =   -647.789  mm,	Z =   -251.487  mm,
	W =  90.000 deg,	P =   0.000 deg,	R =   90.000 deg
};
P[2852]{
   GP1:
	UF : 0, UT : 6,		CONFIG : 'N U T, 0, 0, 0',
	X =  111.225  mm,	Y =   -647.338  mm,	Z =   -251.074  mm,
	W =  90.000 deg,	P =   0.000 deg,	R =   90.000 deg
};
P[2853]{
   GP1:
	UF : 0, UT : 6,		CONFIG : 'N U T, 0, 0, 0',
	X =  112.254  mm,	Y =   -646.639  mm,	Z =   -251.329  mm,
	W =  90.000 deg,	P =   0.000 deg,	R =   90.000 deg
};
P[2854]{
   GP1:
	UF : 0, UT : 6,		CONFIG : 'N U T, 0, 0, 0',
	X =  112.958  mm,	Y =   -646.341  mm,	Z =   -251.066  mm,
	W =  90.000 deg,	P =   0.000 deg,	R =   90.000 deg
};
P[2855]{
   GP1:
	UF : 0, UT : 6,		CONFIG : 'N U T, 0, 0, 0',
	X =  124.694  mm,	Y =   -639.564  mm,	Z =   -251.067  mm,
	W =  90.000 deg,	P =   0.000 deg,	R =   90.000 deg
};
P[2856]{
   GP1:
	UF : 0, UT : 6,		CONFIG : 'N U T, 0, 0, 0',
	X =  129.432  mm,	Y =   -636.794  mm,	Z =   -251.150  mm,
	W =  90.000 deg,	P =   0.000 deg,	R =   90.000 deg
};
P[2857]{
   GP1:
	UF : 0, UT : 6,		CONFIG : 'N U T, 0, 0, 0',
	X =  133.155  mm,	Y =   -634.576  mm,	Z =   -251.314  mm,
	W =  90.000 deg,	P =   0.000 deg,	R =   90.000 deg
};
P[2858]{
   GP1:
	UF : 0, UT : 6,		CONFIG : 'N U T, 0, 0, 0',
	X =  134.202  mm,	Y =   -633.923  mm,	Z =   -251.432  mm,
	W =  90.000 deg,	P =   0.000 deg,	R =   90.000 deg
};
P[2859]{
   GP1:
	UF : 0, UT : 6,		CONFIG : 'N U T, 0, 0, 0',
	X =  139.199  mm,	Y =   -631.158  mm,	Z =   -251.141  mm,
	W =  90.000 deg,	P =   0.000 deg,	R =   90.000 deg
};
P[2860]{
   GP1:
	UF : 0, UT : 6,		CONFIG : 'N U T, 0, 0, 0',
	X =  143.547  mm,	Y =   -628.511  mm,	Z =   -251.473  mm,
	W =  90.000 deg,	P =   0.000 deg,	R =   90.000 deg
};
P[2861]{
   GP1:
	UF : 0, UT : 6,		CONFIG : 'N U T, 0, 0, 0',
	X =  145.385  mm,	Y =   -627.451  mm,	Z =   -251.470  mm,
	W =  90.000 deg,	P =   0.000 deg,	R =   90.000 deg
};
P[2862]{
   GP1:
	UF : 0, UT : 6,		CONFIG : 'N U T, 0, 0, 0',
	X =  146.198  mm,	Y =   -627.021  mm,	Z =   -251.374  mm,
	W =  90.000 deg,	P =   0.000 deg,	R =   90.000 deg
};
P[2863]{
   GP1:
	UF : 0, UT : 6,		CONFIG : 'N U T, 0, 0, 0',
	X =  148.444  mm,	Y =   -625.671  mm,	Z =   -251.505  mm,
	W =  90.000 deg,	P =   0.000 deg,	R =   90.000 deg
};
P[2864]{
   GP1:
	UF : 0, UT : 6,		CONFIG : 'N U T, 0, 0, 0',
	X =  151.895  mm,	Y =   -623.782  mm,	Z =   -251.252  mm,
	W =  90.000 deg,	P =   0.000 deg,	R =   90.000 deg
};
P[2865]{
   GP1:
	UF : 0, UT : 6,		CONFIG : 'N U T, 0, 0, 0',
	X =  154.530  mm,	Y =   -622.201  mm,	Z =   -251.398  mm,
	W =  90.000 deg,	P =   0.000 deg,	R =   90.000 deg
};
P[2866]{
   GP1:
	UF : 0, UT : 6,		CONFIG : 'N U T, 0, 0, 0',
	X =  155.472  mm,	Y =   -621.701  mm,	Z =   -251.291  mm,
	W =  90.000 deg,	P =   0.000 deg,	R =   90.000 deg
};
P[2867]{
   GP1:
	UF : 0, UT : 6,		CONFIG : 'N U T, 0, 0, 0',
	X =  157.309  mm,	Y =   -620.675  mm,	Z =   -251.206  mm,
	W =  90.000 deg,	P =   0.000 deg,	R =   90.000 deg
};
P[2868]{
   GP1:
	UF : 0, UT : 6,		CONFIG : 'N U T, 0, 0, 0',
	X =  159.452  mm,	Y =   -619.460  mm,	Z =   -251.153  mm,
	W =  90.000 deg,	P =   0.000 deg,	R =   90.000 deg
};
P[2869]{
   GP1:
	UF : 0, UT : 6,		CONFIG : 'N U T, 0, 0, 0',
	X =  160.368  mm,	Y =   -618.865  mm,	Z =   -251.312  mm,
	W =  90.000 deg,	P =   0.000 deg,	R =   90.000 deg
};
P[2870]{
   GP1:
	UF : 0, UT : 6,		CONFIG : 'N U T, 0, 0, 0',
	X =  163.587  mm,	Y =   -617.078  mm,	Z =   -251.139  mm,
	W =  90.000 deg,	P =   0.000 deg,	R =   90.000 deg
};
P[2871]{
   GP1:
	UF : 0, UT : 6,		CONFIG : 'N U T, 0, 0, 0',
	X =  165.438  mm,	Y =   -615.983  mm,	Z =   -251.201  mm,
	W =  90.000 deg,	P =   0.000 deg,	R =   90.000 deg
};
P[2872]{
   GP1:
	UF : 0, UT : 6,		CONFIG : 'N U T, 0, 0, 0',
	X =  167.235  mm,	Y =   -614.851  mm,	Z =   -251.430  mm,
	W =  90.000 deg,	P =   0.000 deg,	R =   90.000 deg
};
P[2873]{
   GP1:
	UF : 0, UT : 6,		CONFIG : 'N U T, 0, 0, 0',
	X =  169.556  mm,	Y =   -613.513  mm,	Z =   -251.428  mm,
	W =  90.000 deg,	P =   0.000 deg,	R =   90.000 deg
};
P[2874]{
   GP1:
	UF : 0, UT : 6,		CONFIG : 'N U T, 0, 0, 0',
	X =  170.199  mm,	Y =   -613.213  mm,	Z =   -251.255  mm,
	W =  90.000 deg,	P =   0.000 deg,	R =   90.000 deg
};
P[2875]{
   GP1:
	UF : 0, UT : 6,		CONFIG : 'N U T, 0, 0, 0',
	X =  172.457  mm,	Y =   -611.981  mm,	Z =   -251.079  mm,
	W =  90.000 deg,	P =   0.000 deg,	R =   90.000 deg
};
P[2876]{
   GP1:
	UF : 0, UT : 6,		CONFIG : 'N U T, 0, 0, 0',
	X =  174.587  mm,	Y =   -610.594  mm,	Z =   -251.459  mm,
	W =  90.000 deg,	P =   0.000 deg,	R =   90.000 deg
};
P[2877]{
   GP1:
	UF : 0, UT : 6,		CONFIG : 'N U T, 0, 0, 0',
	X =  175.338  mm,	Y =   -610.329  mm,	Z =   -251.051  mm,
	W =  90.000 deg,	P =   0.000 deg,	R =   90.000 deg
};
P[2878]{
   GP1:
	UF : 0, UT : 6,		CONFIG : 'N U T, 0, 0, 0',
	X =  178.247  mm,	Y =   -608.545  mm,	Z =   -251.305  mm,
	W =  90.000 deg,	P =   0.000 deg,	R =   90.000 deg
};
P[2879]{
   GP1:
	UF : 0, UT : 6,		CONFIG : 'N U T, 0, 0, 0',
	X =  178.919  mm,	Y =   -608.248  mm,	Z =   -251.085  mm,
	W =  90.000 deg,	P =   0.000 deg,	R =   90.000 deg
};
P[2880]{
   GP1:
	UF : 0, UT : 6,		CONFIG : 'N U T, 0, 0, 0',
	X =  180.705  mm,	Y =   -607.087  mm,	Z =   -251.398  mm,
	W =  90.000 deg,	P =   0.000 deg,	R =   90.000 deg
};
P[2881]{
   GP1:
	UF : 0, UT : 6,		CONFIG : 'N U T, 0, 0, 0',
	X =  182.372  mm,	Y =   -606.217  mm,	Z =   -251.176  mm,
	W =  90.000 deg,	P =   0.000 deg,	R =   90.000 deg
};
P[2882]{
   GP1:
	UF : 0, UT : 6,		CONFIG : 'N U T, 0, 0, 0',
	X =  183.552  mm,	Y =   -605.521  mm,	Z =   -251.212  mm,
	W =  90.000 deg,	P =   0.000 deg,	R =   90.000 deg
};
P[2883]{
   GP1:
	UF : 0, UT : 6,		CONFIG : 'N U T, 0, 0, 0',
	X =  184.884  mm,	Y =   -604.665  mm,	Z =   -251.422  mm,
	W =  90.000 deg,	P =   0.000 deg,	R =   90.000 deg
};
P[2884]{
   GP1:
	UF : 0, UT : 6,		CONFIG : 'N U T, 0, 0, 0',
	X =  186.046  mm,	Y =   -604.027  mm,	Z =   -251.340  mm,
	W =  90.000 deg,	P =   0.000 deg,	R =   90.000 deg
};
P[2885]{
   GP1:
	UF : 0, UT : 6,		CONFIG : 'N U T, 0, 0, 0',
	X =  188.896  mm,	Y =   -602.386  mm,	Z =   -251.330  mm,
	W =  90.000 deg,	P =   0.000 deg,	R =   90.000 deg
};
P[2886]{
   GP1:
	UF : 0, UT : 6,		CONFIG : 'N U T, 0, 0, 0',
	X =  190.734  mm,	Y =   -601.399  mm,	Z =   -251.152  mm,
	W =  90.000 deg,	P =   0.000 deg,	R =   90.000 deg
};
P[2887]{
   GP1:
	UF : 0, UT : 6,		CONFIG : 'N U T, 0, 0, 0',
	X =  193.103  mm,	Y =   -599.901  mm,	Z =   -251.465  mm,
	W =  90.000 deg,	P =   0.000 deg,	R =   90.000 deg
};
P[2888]{
   GP1:
	UF : 0, UT : 6,		CONFIG : 'N U T, 0, 0, 0',
	X =  194.069  mm,	Y =   -599.471  mm,	Z =   -251.155  mm,
	W =  90.000 deg,	P =   0.000 deg,	R =   90.000 deg
};
P[2889]{
   GP1:
	UF : 0, UT : 6,		CONFIG : 'N U T, 0, 0, 0',
	X =  195.259  mm,	Y =   -598.839  mm,	Z =   -251.021  mm,
	W =  90.000 deg,	P =   0.000 deg,	R =   90.000 deg
};
P[2890]{
   GP1:
	UF : 0, UT : 6,		CONFIG : 'N U T, 0, 0, 0',
	X =  196.350  mm,	Y =   -598.209  mm,	Z =   -251.022  mm,
	W =  90.000 deg,	P =   0.000 deg,	R =   90.000 deg
};
P[2891]{
   GP1:
	UF : 0, UT : 6,		CONFIG : 'N U T, 0, 0, 0',
	X =  203.115  mm,	Y =   -594.190  mm,	Z =   -251.296  mm,
	W =  90.000 deg,	P =   0.000 deg,	R =   90.000 deg
};
P[2892]{
   GP1:
	UF : 0, UT : 6,		CONFIG : 'N U T, 0, 0, 0',
	X =  209.718  mm,	Y =   -590.303  mm,	Z =   -251.477  mm,
	W =  90.000 deg,	P =   0.000 deg,	R =   90.000 deg
};
P[2893]{
   GP1:
	UF : 0, UT : 6,		CONFIG : 'N U T, 0, 0, 0',
	X =  210.641  mm,	Y =   -589.763  mm,	Z =   -251.494  mm,
	W =  90.000 deg,	P =   0.000 deg,	R =   90.000 deg
};
P[2894]{
   GP1:
	UF : 0, UT : 6,		CONFIG : 'N U T, 0, 0, 0',
	X =  211.542  mm,	Y =   -589.285  mm,	Z =   -251.391  mm,
	W =  90.000 deg,	P =   0.000 deg,	R =   90.000 deg
};
P[2895]{
   GP1:
	UF : 0, UT : 6,		CONFIG : 'N U T, 0, 0, 0',
	X =  213.006  mm,	Y =   -588.439  mm,	Z =   -251.393  mm,
	W =  90.000 deg,	P =   0.000 deg,	R =   90.000 deg
};
P[2896]{
   GP1:
	UF : 0, UT : 6,		CONFIG : 'N U T, 0, 0, 0',
	X =  213.990  mm,	Y =   -587.855  mm,	Z =   -251.432  mm,
	W =  90.000 deg,	P =   0.000 deg,	R =   90.000 deg
};
P[2897]{
   GP1:
	UF : 0, UT : 6,		CONFIG : 'N U T, 0, 0, 0',
	X =  216.991  mm,	Y =   -586.238  mm,	Z =   -251.150  mm,
	W =  90.000 deg,	P =   0.000 deg,	R =   90.000 deg
};
P[2898]{
   GP1:
	UF : 0, UT : 6,		CONFIG : 'N U T, 0, 0, 0',
	X =  218.362  mm,	Y =   -585.476  mm,	Z =   -251.080  mm,
	W =  90.000 deg,	P =   0.000 deg,	R =   90.000 deg
};
P[2899]{
   GP1:
	UF : 0, UT : 6,		CONFIG : 'N U T, 0, 0, 0',
	X =  220.942  mm,	Y =   -583.867  mm,	Z =   -251.366  mm,
	W =  90.000 deg,	P =   0.000 deg,	R =   90.000 deg
};
P[2900]{
   GP1:
	UF : 0, UT : 6,		CONFIG : 'N U T, 0, 0, 0',
	X =  221.618  mm,	Y =   -583.506  mm,	Z =   -251.298  mm,
	W =  90.000 deg,	P =   0.000 deg,	R =   90.000 deg
};
P[2901]{
   GP1:
	UF : 0, UT : 6,		CONFIG : 'N U T, 0, 0, 0',
	X =  223.093  mm,	Y =   -582.590  mm,	Z =   -251.453  mm,
	W =  90.000 deg,	P =   0.000 deg,	R =   90.000 deg
};
P[2902]{
   GP1:
	UF : 0, UT : 6,		CONFIG : 'N U T, 0, 0, 0',
	X =  224.850  mm,	Y =   -581.555  mm,	Z =   -251.502  mm,
	W =  90.000 deg,	P =   0.000 deg,	R =   90.000 deg
};
P[2903]{
   GP1:
	UF : 0, UT : 6,		CONFIG : 'N U T, 0, 0, 0',
	X =  226.605  mm,	Y =   -580.684  mm,	Z =   -251.157  mm,
	W =  90.000 deg,	P =   0.000 deg,	R =   90.000 deg
};
P[2904]{
   GP1:
	UF : 0, UT : 6,		CONFIG : 'N U T, 0, 0, 0',
	X =  227.954  mm,	Y =   -579.933  mm,	Z =   -251.090  mm,
	W =  90.000 deg,	P =   0.000 deg,	R =   90.000 deg
};
P[2905]{
   GP1:
	UF : 0, UT : 6,		CONFIG : 'N U T, 0, 0, 0',
	X =  229.059  mm,	Y =   -579.147  mm,	Z =   -251.449  mm,
	W =  90.000 deg,	P =   0.000 deg,	R =   90.000 deg
};
P[2906]{
   GP1:
	UF : 0, UT : 6,		CONFIG : 'N U T, 0, 0, 0',
	X =  231.542  mm,	Y =   -577.809  mm,	Z =   -251.220  mm,
	W =  90.000 deg,	P =   0.000 deg,	R =   90.000 deg
};
P[2907]{
   GP1:
	UF : 0, UT : 6,		CONFIG : 'N U T, 0, 0, 0',
	X =  232.891  mm,	Y =   -576.930  mm,	Z =   -251.459  mm,
	W =  90.000 deg,	P =   0.000 deg,	R =   90.000 deg
};
P[2908]{
   GP1:
	UF : 0, UT : 6,		CONFIG : 'N U T, 0, 0, 0',
	X =  236.360  mm,	Y =   -575.020  mm,	Z =   -251.234  mm,
	W =  90.000 deg,	P =   0.000 deg,	R =   90.000 deg
};
P[2909]{
   GP1:
	UF : 0, UT : 6,		CONFIG : 'N U T, 0, 0, 0',
	X =  241.110  mm,	Y =   -572.227  mm,	Z =   -251.357  mm,
	W =  90.000 deg,	P =   0.000 deg,	R =   90.000 deg
};
P[2910]{
   GP1:
	UF : 0, UT : 6,		CONFIG : 'N U T, 0, 0, 0',
	X =  242.180  mm,	Y =   -571.559  mm,	Z =   -251.479  mm,
	W =  90.000 deg,	P =   0.000 deg,	R =   90.000 deg
};
P[2911]{
   GP1:
	UF : 0, UT : 6,		CONFIG : 'N U T, 0, 0, 0',
	X =  244.999  mm,	Y =   -569.949  mm,	Z =   -251.435  mm,
	W =  90.000 deg,	P =   0.000 deg,	R =   90.000 deg
};
P[2912]{
   GP1:
	UF : 0, UT : 6,		CONFIG : 'N U T, 0, 0, 0',
	X =  247.045  mm,	Y =   -568.803  mm,	Z =   -251.351  mm,
	W =  90.000 deg,	P =   0.000 deg,	R =   90.000 deg
};
P[2913]{
   GP1:
	UF : 0, UT : 6,		CONFIG : 'N U T, 0, 0, 0',
	X =  247.833  mm,	Y =   -568.352  mm,	Z =   -251.340  mm,
	W =  90.000 deg,	P =   0.000 deg,	R =   90.000 deg
};
P[2914]{
   GP1:
	UF : 0, UT : 6,		CONFIG : 'N U T, 0, 0, 0',
	X =  250.224  mm,	Y =   -567.044  mm,	Z =   -251.165  mm,
	W =  90.000 deg,	P =   0.000 deg,	R =   90.000 deg
};
P[2915]{
   GP1:
	UF : 0, UT : 6,		CONFIG : 'N U T, 0, 0, 0',
	X =  251.401  mm,	Y =   -566.273  mm,	Z =   -251.386  mm,
	W =  90.000 deg,	P =   0.000 deg,	R =   90.000 deg
};
P[2916]{
   GP1:
	UF : 0, UT : 6,		CONFIG : 'N U T, 0, 0, 0',
	X =  254.843  mm,	Y =   -564.277  mm,	Z =   -251.408  mm,
	W =  90.000 deg,	P =   0.000 deg,	R =   90.000 deg
};
P[2917]{
   GP1:
	UF : 0, UT : 6,		CONFIG : 'N U T, 0, 0, 0',
	X =  256.795  mm,	Y =   -563.204  mm,	Z =   -251.275  mm,
	W =  90.000 deg,	P =   0.000 deg,	R =   90.000 deg
};
P[2918]{
   GP1:
	UF : 0, UT : 6,		CONFIG : 'N U T, 0, 0, 0',
	X =  258.604  mm,	Y =   -562.089  mm,	Z =   -251.447  mm,
	W =  90.000 deg,	P =   0.000 deg,	R =   90.000 deg
};
P[2919]{
   GP1:
	UF : 0, UT : 6,		CONFIG : 'N U T, 0, 0, 0',
	X =  260.095  mm,	Y =   -561.240  mm,	Z =   -251.417  mm,
	W =  90.000 deg,	P =   0.000 deg,	R =   90.000 deg
};
P[2920]{
   GP1:
	UF : 0, UT : 6,		CONFIG : 'N U T, 0, 0, 0',
	X =  265.317  mm,	Y =   -558.255  mm,	Z =   -251.345  mm,
	W =  90.000 deg,	P =   0.000 deg,	R =   90.000 deg
};
P[2921]{
   GP1:
	UF : 0, UT : 6,		CONFIG : 'N U T, 0, 0, 0',
	X =  266.261  mm,	Y =   -557.838  mm,	Z =   -251.036  mm,
	W =  90.000 deg,	P =   0.000 deg,	R =   90.000 deg
};
P[2922]{
   GP1:
	UF : 0, UT : 6,		CONFIG : 'N U T, 0, 0, 0',
	X =  269.626  mm,	Y =   -555.767  mm,	Z =   -251.345  mm,
	W =  90.000 deg,	P =   0.000 deg,	R =   90.000 deg
};
P[2923]{
   GP1:
	UF : 0, UT : 6,		CONFIG : 'N U T, 0, 0, 0',
	X =  272.189  mm,	Y =   -554.366  mm,	Z =   -251.153  mm,
	W =  90.000 deg,	P =   0.000 deg,	R =   90.000 deg
};
P[2924]{
   GP1:
	UF : 0, UT : 6,		CONFIG : 'N U T, 0, 0, 0',
	X =  274.866  mm,	Y =   -552.702  mm,	Z =   -251.441  mm,
	W =  90.000 deg,	P =   0.000 deg,	R =   90.000 deg
};
P[2925]{
   GP1:
	UF : 0, UT : 6,		CONFIG : 'N U T, 0, 0, 0',
	X =  281.555  mm,	Y =   -548.821  mm,	Z =   -251.486  mm,
	W =  90.000 deg,	P =   0.000 deg,	R =   90.000 deg
};
P[2926]{
   GP1:
	UF : 0, UT : 6,		CONFIG : 'N U T, 0, 0, 0',
	X =  282.190  mm,	Y =   -548.617  mm,	Z =   -251.093  mm,
	W =  90.000 deg,	P =   0.000 deg,	R =   90.000 deg
};
P[2927]{
   GP1:
	UF : 0, UT : 6,		CONFIG : 'N U T, 0, 0, 0',
	X =  284.211  mm,	Y =   -547.413  mm,	Z =   -251.179  mm,
	W =  90.000 deg,	P =   0.000 deg,	R =   90.000 deg
};
P[2928]{
   GP1:
	UF : 0, UT : 6,		CONFIG : 'N U T, 0, 0, 0',
	X =  284.805  mm,	Y =   -546.994  mm,	Z =   -251.367  mm,
	W =  90.000 deg,	P =   0.000 deg,	R =   90.000 deg
};
P[2929]{
   GP1:
	UF : 0, UT : 6,		CONFIG : 'N U T, 0, 0, 0',
	X =  289.178  mm,	Y =   -544.470  mm,	Z =   -251.364  mm,
	W =  90.000 deg,	P =   0.000 deg,	R =   90.000 deg
};
P[2930]{
   GP1:
	UF : 0, UT : 6,		CONFIG : 'N U T, 0, 0, 0',
	X =  290.282  mm,	Y =   -543.863  mm,	Z =   -251.289  mm,
	W =  90.000 deg,	P =   0.000 deg,	R =   90.000 deg
};
P[2931]{
   GP1:
	UF : 0, UT : 6,		CONFIG : 'N U T, 0, 0, 0',
	X =  294.257  mm,	Y =   -541.664  mm,	Z =   -251.057  mm,
	W =  90.000 deg,	P =   0.000 deg,	R =   90.000 deg
};
P[2932]{
   GP1:
	UF : 0, UT : 6,		CONFIG : 'N U T, 0, 0, 0',
	X =  294.912  mm,	Y =   -541.167  mm,	Z =   -251.346  mm,
	W =  90.000 deg,	P =   0.000 deg,	R =   90.000 deg
};
P[2933]{
   GP1:
	UF : 0, UT : 6,		CONFIG : 'N U T, 0, 0, 0',
	X =  296.022  mm,	Y =   -540.649  mm,	Z =   -251.046  mm,
	W =  90.000 deg,	P =   0.000 deg,	R =   90.000 deg
};
P[2934]{
   GP1:
	UF : 0, UT : 6,		CONFIG : 'N U T, 0, 0, 0',
	X =  297.421  mm,	Y =   -539.808  mm,	Z =   -251.129  mm,
	W =  90.000 deg,	P =   0.000 deg,	R =   90.000 deg
};
P[2935]{
   GP1:
	UF : 0, UT : 6,		CONFIG : 'N U T, 0, 0, 0',
	X =  300.549  mm,	Y =   -537.962  mm,	Z =   -251.224  mm,
	W =  90.000 deg,	P =   0.000 deg,	R =   90.000 deg
};
P[2936]{
   GP1:
	UF : 0, UT : 6,		CONFIG : 'N U T, 0, 0, 0',
	X =  303.330  mm,	Y =   -536.299  mm,	Z =   -251.363  mm,
	W =  90.000 deg,	P =   0.000 deg,	R =   90.000 deg
};
P[2937]{
   GP1:
	UF : 0, UT : 6,		CONFIG : 'N U T, 0, 0, 0',
	X =  304.285  mm,	Y =   -535.792  mm,	Z =   -251.256  mm,
	W =  90.000 deg,	P =   0.000 deg,	R =   90.000 deg
};
P[2938]{
   GP1:
	UF : 0, UT : 6,		CONFIG : 'N U T, 0, 0, 0',
	X =  306.057  mm,	Y =   -534.670  mm,	Z =   -251.495  mm,
	W =  90.000 deg,	P =   0.000 deg,	R =   90.000 deg
};
P[2939]{
   GP1:
	UF : 0, UT : 6,		CONFIG : 'N U T, 0, 0, 0',
	X =  307.108  mm,	Y =   -534.173  mm,	Z =   -251.230  mm,
	W =  90.000 deg,	P =   0.000 deg,	R =   90.000 deg
};
P[2940]{
   GP1:
	UF : 0, UT : 6,		CONFIG : 'N U T, 0, 0, 0',
	X =  308.963  mm,	Y =   -533.165  mm,	Z =   -251.076  mm,
	W =  90.000 deg,	P =   0.000 deg,	R =   90.000 deg
};
P[2941]{
   GP1:
	UF : 0, UT : 6,		CONFIG : 'N U T, 0, 0, 0',
	X =  312.861  mm,	Y =   -530.756  mm,	Z =   -251.461  mm,
	W =  90.000 deg,	P =   0.000 deg,	R =   90.000 deg
};
P[2942]{
   GP1:
	UF : 0, UT : 6,		CONFIG : 'N U T, 0, 0, 0',
	X =  313.930  mm,	Y =   -530.134  mm,	Z =   -251.472  mm,
	W =  90.000 deg,	P =   0.000 deg,	R =   90.000 deg
};
P[2943]{
   GP1:
	UF : 0, UT : 6,		CONFIG : 'N U T, 0, 0, 0',
	X =  316.928  mm,	Y =   -528.428  mm,	Z =   -251.410  mm,
	W =  90.000 deg,	P =   0.000 deg,	R =   90.000 deg
};
P[2944]{
   GP1:
	UF : 0, UT : 6,		CONFIG : 'N U T, 0, 0, 0',
	X =  318.994  mm,	Y =   -527.195  mm,	Z =   -251.507  mm,
	W =  90.000 deg,	P =   0.000 deg,	R =   90.000 deg
};
P[2945]{
   GP1:
	UF : 0, UT : 6,		CONFIG : 'N U T, 0, 0, 0',
	X =  320.877  mm,	Y =   -526.200  mm,	Z =   -251.284  mm,
	W =  90.000 deg,	P =   0.000 deg,	R =   90.000 deg
};
P[2946]{
   GP1:
	UF : 0, UT : 6,		CONFIG : 'N U T, 0, 0, 0',
	X =  322.852  mm,	Y =   -525.132  mm,	Z =   -251.108  mm,
	W =  90.000 deg,	P =   0.000 deg,	R =   90.000 deg
};
P[2947]{
   GP1:
	UF : 0, UT : 6,		CONFIG : 'N U T, 0, 0, 0',
	X =  324.488  mm,	Y =   -524.059  mm,	Z =   -251.421  mm,
	W =  90.000 deg,	P =   0.000 deg,	R =   90.000 deg
};
P[2948]{
   GP1:
	UF : 0, UT : 6,		CONFIG : 'N U T, 0, 0, 0',
	X =  326.523  mm,	Y =   -522.908  mm,	Z =   -251.361  mm,
	W =  90.000 deg,	P =   0.000 deg,	R =   90.000 deg
};
P[2949]{
   GP1:
	UF : 0, UT : 6,		CONFIG : 'N U T, 0, 0, 0',
	X =  327.456  mm,	Y =   -522.349  mm,	Z =   -251.410  mm,
	W =  90.000 deg,	P =   0.000 deg,	R =   90.000 deg
};
P[2950]{
   GP1:
	UF : 0, UT : 6,		CONFIG : 'N U T, 0, 0, 0',
	X =  329.048  mm,	Y =   -521.527  mm,	Z =   -251.176  mm,
	W =  90.000 deg,	P =   0.000 deg,	R =   90.000 deg
};
P[2951]{
   GP1:
	UF : 0, UT : 6,		CONFIG : 'N U T, 0, 0, 0',
	X =  330.315  mm,	Y =   -520.701  mm,	Z =   -251.406  mm,
	W =  90.000 deg,	P =   0.000 deg,	R =   90.000 deg
};
P[2952]{
   GP1:
	UF : 0, UT : 6,		CONFIG : 'N U T, 0, 0, 0',
	X =  332.801  mm,	Y =   -519.401  mm,	Z =   -251.077  mm,
	W =  90.000 deg,	P =   0.000 deg,	R =   90.000 deg
};
P[2953]{
   GP1:
	UF : 0, UT : 6,		CONFIG : 'N U T, 0, 0, 0',
	X =  334.773  mm,	Y =   -518.120  mm,	Z =   -251.421  mm,
	W =  90.000 deg,	P =   0.000 deg,	R =   90.000 deg
};
P[2954]{
   GP1:
	UF : 0, UT : 6,		CONFIG : 'N U T, 0, 0, 0',
	X =  335.697  mm,	Y =   -517.561  mm,	Z =   -251.484  mm,
	W =  90.000 deg,	P =   0.000 deg,	R =   90.000 deg
};
P[2955]{
   GP1:
	UF : 0, UT : 6,		CONFIG : 'N U T, 0, 0, 0',
	X =  336.655  mm,	Y =   -517.016  mm,	Z =   -251.464  mm,
	W =  90.000 deg,	P =   0.000 deg,	R =   90.000 deg
};
P[2956]{
   GP1:
	UF : 0, UT : 6,		CONFIG : 'N U T, 0, 0, 0',
	X =  339.243  mm,	Y =   -515.616  mm,	Z =   -251.235  mm,
	W =  90.000 deg,	P =   0.000 deg,	R =   90.000 deg
};
P[2957]{
   GP1:
	UF : 0, UT : 6,		CONFIG : 'N U T, 0, 0, 0',
	X =  340.458  mm,	Y =   -514.839  mm,	Z =   -251.418  mm,
	W =  90.000 deg,	P =   0.000 deg,	R =   90.000 deg
};
P[2958]{
   GP1:
	UF : 0, UT : 6,		CONFIG : 'N U T, 0, 0, 0',
	X =  341.329  mm,	Y =   -514.397  mm,	Z =   -251.271  mm,
	W =  90.000 deg,	P =   0.000 deg,	R =   90.000 deg
};
P[2959]{
   GP1:
	UF : 0, UT : 6,		CONFIG : 'N U T, 0, 0, 0',
	X =  342.359  mm,	Y =   -513.901  mm,	Z =   -251.029  mm,
	W =  90.000 deg,	P =   0.000 deg,	R =   90.000 deg
};
P[2960]{
   GP1:
	UF : 0, UT : 6,		CONFIG : 'N U T, 0, 0, 0',
	X =  344.773  mm,	Y =   -512.339  mm,	Z =   -251.439  mm,
	W =  90.000 deg,	P =   0.000 deg,	R =   90.000 deg
};
P[2961]{
   GP1:
	UF : 0, UT : 6,		CONFIG : 'N U T, 0, 0, 0',
	X =  348.590  mm,	Y =   -510.228  mm,	Z =   -251.213  mm,
	W =  90.000 deg,	P =   0.000 deg,	R =   90.000 deg
};
P[2962]{
   GP1:
	UF : 0, UT : 6,		CONFIG : 'N U T, 0, 0, 0',
	X =  349.421  mm,	Y =   -509.656  mm,	Z =   -251.437  mm,
	W =  90.000 deg,	P =   0.000 deg,	R =   90.000 deg
};
P[2963]{
   GP1:
	UF : 0, UT : 6,		CONFIG : 'N U T, 0, 0, 0',
	X =  350.325  mm,	Y =   -509.222  mm,	Z =   -251.223  mm,
	W =  90.000 deg,	P =   0.000 deg,	R =   90.000 deg
};
P[2964]{
   GP1:
	UF : 0, UT : 6,		CONFIG : 'N U T, 0, 0, 0',
	X =  354.710  mm,	Y =   -506.730  mm,	Z =   -251.129  mm,
	W =  90.000 deg,	P =   0.000 deg,	R =   90.000 deg
};
P[2965]{
   GP1:
	UF : 0, UT : 6,		CONFIG : 'N U T, 0, 0, 0',
	X =  357.049  mm,	Y =   -505.362  mm,	Z =   -251.169  mm,
	W =  90.000 deg,	P =   0.000 deg,	R =   90.000 deg
};
P[2966]{
   GP1:
	UF : 0, UT : 6,		CONFIG : 'N U T, 0, 0, 0',
	X =  359.894  mm,	Y =   -503.651  mm,	Z =   -251.333  mm,
	W =  90.000 deg,	P =   0.000 deg,	R =   90.000 deg
};
P[2967]{
   GP1:
	UF : 0, UT : 6,		CONFIG : 'N U T, 0, 0, 0',
	X =  362.013  mm,	Y =   -502.494  mm,	Z =   -251.173  mm,
	W =  90.000 deg,	P =   0.000 deg,	R =   90.000 deg
};
P[2968]{
   GP1:
	UF : 0, UT : 6,		CONFIG : 'N U T, 0, 0, 0',
	X =  364.396  mm,	Y =   -501.107  mm,	Z =   -251.203  mm,
	W =  90.000 deg,	P =   0.000 deg,	R =   90.000 deg
};
P[2969]{
   GP1:
	UF : 0, UT : 6,		CONFIG : 'N U T, 0, 0, 0',
	X =  365.110  mm,	Y =   -500.604  mm,	Z =   -251.422  mm,
	W =  90.000 deg,	P =   0.000 deg,	R =   90.000 deg
};
P[2970]{
   GP1:
	UF : 0, UT : 6,		CONFIG : 'N U T, 0, 0, 0',
	X =  366.340  mm,	Y =   -499.959  mm,	Z =   -251.262  mm,
	W =  90.000 deg,	P =   0.000 deg,	R =   90.000 deg
};
P[2971]{
   GP1:
	UF : 0, UT : 6,		CONFIG : 'N U T, 0, 0, 0',
	X =  371.719  mm,	Y =   -496.822  mm,	Z =   -251.340  mm,
	W =  90.000 deg,	P =   0.000 deg,	R =   90.000 deg
};
P[2972]{
   GP1:
	UF : 0, UT : 6,		CONFIG : 'N U T, 0, 0, 0',
	X =  374.009  mm,	Y =   -495.563  mm,	Z =   -251.185  mm,
	W =  90.000 deg,	P =   0.000 deg,	R =   90.000 deg
};
P[2973]{
   GP1:
	UF : 0, UT : 6,		CONFIG : 'N U T, 0, 0, 0',
	X =  376.667  mm,	Y =   -494.048  mm,	Z =   -251.137  mm,
	W =  90.000 deg,	P =   0.000 deg,	R =   90.000 deg
};
P[2974]{
   GP1:
	UF : 0, UT : 6,		CONFIG : 'N U T, 0, 0, 0',
	X =  384.212  mm,	Y =   -489.580  mm,	Z =   -251.409  mm,
	W =  90.000 deg,	P =   0.000 deg,	R =   90.000 deg
};
P[2975]{
   GP1:
	UF : 0, UT : 6,		CONFIG : 'N U T, 0, 0, 0',
	X =  385.099  mm,	Y =   -489.029  mm,	Z =   -251.504  mm,
	W =  90.000 deg,	P =   0.000 deg,	R =   90.000 deg
};
P[2976]{
   GP1:
	UF : 0, UT : 6,		CONFIG : 'N U T, 0, 0, 0',
	X =  386.533  mm,	Y =   -488.242  mm,	Z =   -251.403  mm,
	W =  90.000 deg,	P =   0.000 deg,	R =   90.000 deg
};
P[2977]{
   GP1:
	UF : 0, UT : 6,		CONFIG : 'N U T, 0, 0, 0',
	X =  388.921  mm,	Y =   -486.948  mm,	Z =   -251.196  mm,
	W =  90.000 deg,	P =   0.000 deg,	R =   90.000 deg
};
P[2978]{
   GP1:
	UF : 0, UT : 6,		CONFIG : 'N U T, 0, 0, 0',
	X =  391.104  mm,	Y =   -485.695  mm,	Z =   -251.181  mm,
	W =  90.000 deg,	P =   0.000 deg,	R =   90.000 deg
};
P[2979]{
   GP1:
	UF : 0, UT : 6,		CONFIG : 'N U T, 0, 0, 0',
	X =  392.827  mm,	Y =   -484.584  mm,	Z =   -251.459  mm,
	W =  90.000 deg,	P =   0.000 deg,	R =   90.000 deg
};
P[2980]{
   GP1:
	UF : 0, UT : 6,		CONFIG : 'N U T, 0, 0, 0',
	X =  393.443  mm,	Y =   -484.360  mm,	Z =   -251.143  mm,
	W =  90.000 deg,	P =   0.000 deg,	R =   90.000 deg
};
P[2981]{
   GP1:
	UF : 0, UT : 6,		CONFIG : 'N U T, 0, 0, 0',
	X =  394.111  mm,	Y =   -483.915  mm,	Z =   -251.284  mm,
	W =  90.000 deg,	P =   0.000 deg,	R =   90.000 deg
};
P[2982]{
   GP1:
	UF : 0, UT : 6,		CONFIG : 'N U T, 0, 0, 0',
	X =  394.948  mm,	Y =   -483.418  mm,	Z =   -251.318  mm,
	W =  90.000 deg,	P =   0.000 deg,	R =   90.000 deg
};
P[2983]{
   GP1:
	UF : 0, UT : 6,		CONFIG : 'N U T, 0, 0, 0',
	X =  395.774  mm,	Y =   -482.964  mm,	Z =   -251.264  mm,
	W =  90.000 deg,	P =   0.000 deg,	R =   90.000 deg
};
P[2984]{
   GP1:
	UF : 0, UT : 6,		CONFIG : 'N U T, 0, 0, 0',
	X =  396.916  mm,	Y =   -482.290  mm,	Z =   -251.300  mm,
	W =  90.000 deg,	P =   0.000 deg,	R =   90.000 deg
};
P[2985]{
   GP1:
	UF : 0, UT : 6,		CONFIG : 'N U T, 0, 0, 0',
	X =  398.511  mm,	Y =   -481.342  mm,	Z =   -251.363  mm,
	W =  90.000 deg,	P =   0.000 deg,	R =   90.000 deg
};
P[2986]{
   GP1:
	UF : 0, UT : 6,		CONFIG : 'N U T, 0, 0, 0',
	X =  399.542  mm,	Y =   -480.853  mm,	Z =   -251.105  mm,
	W =  90.000 deg,	P =   0.000 deg,	R =   90.000 deg
};
P[2987]{
   GP1:
	UF : 0, UT : 6,		CONFIG : 'N U T, 0, 0, 0',
	X =  401.428  mm,	Y =   -479.621  mm,	Z =   -251.451  mm,
	W =  90.000 deg,	P =   0.000 deg,	R =   90.000 deg
};
P[2988]{
   GP1:
	UF : 0, UT : 6,		CONFIG : 'N U T, 0, 0, 0',
	X =  402.190  mm,	Y =   -479.184  mm,	Z =   -251.447  mm,
	W =  90.000 deg,	P =   0.000 deg,	R =   90.000 deg
};
P[2989]{
   GP1:
	UF : 0, UT : 6,		CONFIG : 'N U T, 0, 0, 0',
	X =  403.862  mm,	Y =   -478.326  mm,	Z =   -251.184  mm,
	W =  90.000 deg,	P =   0.000 deg,	R =   90.000 deg
};
P[2990]{
   GP1:
	UF : 0, UT : 6,		CONFIG : 'N U T, 0, 0, 0',
	X =  406.339  mm,	Y =   -476.857  mm,	Z =   -251.280  mm,
	W =  90.000 deg,	P =   0.000 deg,	R =   90.000 deg
};
P[2991]{
   GP1:
	UF : 0, UT : 6,		CONFIG : 'N U T, 0, 0, 0',
	X =  407.320  mm,	Y =   -476.373  mm,	Z =   -251.078  mm,
	W =  90.000 deg,	P =   0.000 deg,	R =   90.000 deg
};
P[2992]{
   GP1:
	UF : 0, UT : 6,		CONFIG : 'N U T, 0, 0, 0',
	X =  408.488  mm,	Y =   -475.523  mm,	Z =   -251.506  mm,
	W =  90.000 deg,	P =   0.000 deg,	R =   90.000 deg
};
P[2993]{
   GP1:
	UF : 0, UT : 6,		CONFIG : 'N U T, 0, 0, 0',
	X =  412.713  mm,	Y =   -473.084  mm,	Z =   -251.505  mm,
	W =  90.000 deg,	P =   0.000 deg,	R =   90.000 deg
};
P[2994]{
   GP1:
	UF : 0, UT : 6,		CONFIG : 'N U T, 0, 0, 0',
	X =  413.604  mm,	Y =   -472.575  mm,	Z =   -251.490  mm,
	W =  90.000 deg,	P =   0.000 deg,	R =   90.000 deg
};
P[2995]{
   GP1:
	UF : 0, UT : 6,		CONFIG : 'N U T, 0, 0, 0',
	X =  414.874  mm,	Y =   -471.914  mm,	Z =   -251.314  mm,
	W =  90.000 deg,	P =   0.000 deg,	R =   90.000 deg
};
P[2996]{
   GP1:
	UF : 0, UT : 6,		CONFIG : 'N U T, 0, 0, 0',
	X =  417.976  mm,	Y =   -470.077  mm,	Z =   -251.428  mm,
	W =  90.000 deg,	P =   0.000 deg,	R =   90.000 deg
};
P[2997]{
   GP1:
	UF : 0, UT : 6,		CONFIG : 'N U T, 0, 0, 0',
	X =  419.780  mm,	Y =   -469.061  mm,	Z =   -251.364  mm,
	W =  90.000 deg,	P =   0.000 deg,	R =   90.000 deg
};
P[2998]{
   GP1:
	UF : 0, UT : 6,		CONFIG : 'N U T, 0, 0, 0',
	X =  422.751  mm,	Y =   -467.447  mm,	Z =   -251.117  mm,
	W =  90.000 deg,	P =   0.000 deg,	R =   90.000 deg
};
P[2999]{
   GP1:
	UF : 0, UT : 6,		CONFIG : 'N U T, 0, 0, 0',
	X =  424.402  mm,	Y =   -466.371  mm,	Z =   -251.417  mm,
	W =  90.000 deg,	P =   0.000 deg,	R =   90.000 deg
};
P[3000]{
   GP1:
	UF : 0, UT : 6,		CONFIG : 'N U T, 0, 0, 0',
	X =  425.368  mm,	Y =   -465.890  mm,	Z =   -251.229  mm,
	W =  90.000 deg,	P =   0.000 deg,	R =   90.000 deg
};
P[3001]{
   GP1:
	UF : 0, UT : 6,		CONFIG : 'N U T, 0, 0, 0',
	X =  426.382  mm,	Y =   -465.370  mm,	Z =   -251.070  mm,
	W =  90.000 deg,	P =   0.000 deg,	R =   90.000 deg
};
P[3002]{
   GP1:
	UF : 0, UT : 6,		CONFIG : 'N U T, 0, 0, 0',
	X =  429.751  mm,	Y =   -463.290  mm,	Z =   -251.399  mm,
	W =  90.000 deg,	P =   0.000 deg,	R =   90.000 deg
};
P[3003]{
   GP1:
	UF : 0, UT : 6,		CONFIG : 'N U T, 0, 0, 0',
	X =  431.813  mm,	Y =   -462.205  mm,	Z =   -251.141  mm,
	W =  90.000 deg,	P =   0.000 deg,	R =   90.000 deg
};
P[3004]{
   GP1:
	UF : 0, UT : 6,		CONFIG : 'N U T, 0, 0, 0',
	X =  432.444  mm,	Y =   -461.735  mm,	Z =   -251.398  mm,
	W =  90.000 deg,	P =   0.000 deg,	R =   90.000 deg
};
P[3005]{
   GP1:
	UF : 0, UT : 6,		CONFIG : 'N U T, 0, 0, 0',
	X =  433.185  mm,	Y =   -461.457  mm,	Z =   -251.034  mm,
	W =  90.000 deg,	P =   0.000 deg,	R =   90.000 deg
};
P[3006]{
   GP1:
	UF : 0, UT : 6,		CONFIG : 'N U T, 0, 0, 0',
	X =  435.720  mm,	Y =   -459.817  mm,	Z =   -251.464  mm,
	W =  90.000 deg,	P =   0.000 deg,	R =   90.000 deg
};
P[3007]{
   GP1:
	UF : 0, UT : 6,		CONFIG : 'N U T, 0, 0, 0',
	X =  436.642  mm,	Y =   -459.294  mm,	Z =   -251.440  mm,
	W =  90.000 deg,	P =   0.000 deg,	R =   90.000 deg
};
P[3008]{
   GP1:
	UF : 0, UT : 6,		CONFIG : 'N U T, 0, 0, 0',
	X =  438.191  mm,	Y =   -458.476  mm,	Z =   -251.255  mm,
	W =  90.000 deg,	P =   0.000 deg,	R =   90.000 deg
};
P[3009]{
   GP1:
	UF : 0, UT : 6,		CONFIG : 'N U T, 0, 0, 0',
	X =  440.977  mm,	Y =   -456.880  mm,	Z =   -251.223  mm,
	W =  90.000 deg,	P =   0.000 deg,	R =   90.000 deg
};
P[3010]{
   GP1:
	UF : 0, UT : 6,		CONFIG : 'N U T, 0, 0, 0',
	X =  442.019  mm,	Y =   -456.205  mm,	Z =   -251.403  mm,
	W =  90.000 deg,	P =   0.000 deg,	R =   90.000 deg
};
P[3011]{
   GP1:
	UF : 0, UT : 6,		CONFIG : 'N U T, 0, 0, 0',
	X =  442.936  mm,	Y =   -455.657  mm,	Z =   -251.450  mm,
	W =  90.000 deg,	P =   0.000 deg,	R =   90.000 deg
};
P[3012]{
   GP1:
	UF : 0, UT : 6,		CONFIG : 'N U T, 0, 0, 0',
	X =  443.591  mm,	Y =   -455.284  mm,	Z =   -251.436  mm,
	W =  90.000 deg,	P =   0.000 deg,	R =   90.000 deg
};
P[3013]{
   GP1:
	UF : 0, UT : 6,		CONFIG : 'N U T, 0, 0, 0',
	X =  444.314  mm,	Y =   -454.884  mm,	Z =   -251.392  mm,
	W =  90.000 deg,	P =   0.000 deg,	R =   90.000 deg
};
P[3014]{
   GP1:
	UF : 0, UT : 6,		CONFIG : 'N U T, 0, 0, 0',
	X =  445.511  mm,	Y =   -454.291  mm,	Z =   -251.155  mm,
	W =  90.000 deg,	P =   0.000 deg,	R =   90.000 deg
};
P[3015]{
   GP1:
	UF : 0, UT : 6,		CONFIG : 'N U T, 0, 0, 0',
	X =  447.204  mm,	Y =   -453.192  mm,	Z =   -251.450  mm,
	W =  90.000 deg,	P =   0.000 deg,	R =   90.000 deg
};
P[3016]{
   GP1:
	UF : 0, UT : 6,		CONFIG : 'N U T, 0, 0, 0',
	X =  448.524  mm,	Y =   -452.432  mm,	Z =   -251.445  mm,
	W =  90.000 deg,	P =   0.000 deg,	R =   90.000 deg
};
P[3017]{
   GP1:
	UF : 0, UT : 6,		CONFIG : 'N U T, 0, 0, 0',
	X =  450.215  mm,	Y =   -451.570  mm,	Z =   -251.167  mm,
	W =  90.000 deg,	P =   0.000 deg,	R =   90.000 deg
};
P[3018]{
   GP1:
	UF : 0, UT : 6,		CONFIG : 'N U T, 0, 0, 0',
	X =  456.044  mm,	Y =   -448.085  mm,	Z =   -251.457  mm,
	W =  90.000 deg,	P =   0.000 deg,	R =   90.000 deg
};
P[3019]{
   GP1:
	UF : 0, UT : 6,		CONFIG : 'N U T, 0, 0, 0',
	X =  458.665  mm,	Y =   -446.699  mm,	Z =   -251.146  mm,
	W =  90.000 deg,	P =   0.000 deg,	R =   90.000 deg
};
P[3020]{
   GP1:
	UF : 0, UT : 6,		CONFIG : 'N U T, 0, 0, 0',
	X =  460.415  mm,	Y =   -445.673  mm,	Z =   -251.186  mm,
	W =  90.000 deg,	P =   0.000 deg,	R =   90.000 deg
};
P[3021]{
   GP1:
	UF : 0, UT : 6,		CONFIG : 'N U T, 0, 0, 0',
	X =  461.055  mm,	Y =   -445.240  mm,	Z =   -251.339  mm,
	W =  90.000 deg,	P =   0.000 deg,	R =   90.000 deg
};
P[3022]{
   GP1:
	UF : 0, UT : 6,		CONFIG : 'N U T, 0, 0, 0',
	X =  463.189  mm,	Y =   -443.996  mm,	Z =   -251.368  mm,
	W =  90.000 deg,	P =   0.000 deg,	R =   90.000 deg
};
P[3023]{
   GP1:
	UF : 0, UT : 6,		CONFIG : 'N U T, 0, 0, 0',
	X =  463.828  mm,	Y =   -443.629  mm,	Z =   -251.361  mm,
	W =  90.000 deg,	P =   0.000 deg,	R =   90.000 deg
};
P[3024]{
   GP1:
	UF : 0, UT : 6,		CONFIG : 'N U T, 0, 0, 0',
	X =  466.269  mm,	Y =   -442.179  mm,	Z =   -251.461  mm,
	W =  90.000 deg,	P =   0.000 deg,	R =   90.000 deg
};
P[3025]{
   GP1:
	UF : 0, UT : 6,		CONFIG : 'N U T, 0, 0, 0',
	X =  467.416  mm,	Y =   -441.598  mm,	Z =   -251.264  mm,
	W =  90.000 deg,	P =   0.000 deg,	R =   90.000 deg
};
P[3026]{
   GP1:
	UF : 0, UT : 6,		CONFIG : 'N U T, 0, 0, 0',
	X =  468.766  mm,	Y =   -440.879  mm,	Z =   -251.119  mm,
	W =  90.000 deg,	P =   0.000 deg,	R =   90.000 deg
};
P[3027]{
   GP1:
	UF : 0, UT : 6,		CONFIG : 'N U T, 0, 0, 0',
	X =  472.321  mm,	Y =   -438.766  mm,	Z =   -251.264  mm,
	W =  90.000 deg,	P =   0.000 deg,	R =   90.000 deg
};
P[3028]{
   GP1:
	UF : 0, UT : 6,		CONFIG : 'N U T, 0, 0, 0',
	X =  474.152  mm,	Y =   -437.669  mm,	Z =   -251.359  mm,
	W =  90.000 deg,	P =   0.000 deg,	R =   90.000 deg
};
P[3029]{
   GP1:
	UF : 0, UT : 6,		CONFIG : 'N U T, 0, 0, 0',
	X =  476.461  mm,	Y =   -436.304  mm,	Z =   -251.440  mm,
	W =  90.000 deg,	P =   0.000 deg,	R =   90.000 deg
};
P[3030]{
   GP1:
	UF : 0, UT : 6,		CONFIG : 'N U T, 0, 0, 0',
	X =  478.394  mm,	Y =   -435.358  mm,	Z =   -251.023  mm,
	W =  90.000 deg,	P =   0.000 deg,	R =   90.000 deg
};
P[3031]{
   GP1:
	UF : 0, UT : 6,		CONFIG : 'N U T, 0, 0, 0',
	X =  479.632  mm,	Y =   -434.478  mm,	Z =   -251.424  mm,
	W =  90.000 deg,	P =   0.000 deg,	R =   90.000 deg
};
P[3032]{
   GP1:
	UF : 0, UT : 6,		CONFIG : 'N U T, 0, 0, 0',
	X =  480.613  mm,	Y =   -433.911  mm,	Z =   -251.425  mm,
	W =  90.000 deg,	P =   0.000 deg,	R =   90.000 deg
};
P[3033]{
   GP1:
	UF : 0, UT : 6,		CONFIG : 'N U T, 0, 0, 0',
	X =  484.619  mm,	Y =   -431.625  mm,	Z =   -251.361  mm,
	W =  90.000 deg,	P =   0.000 deg,	R =   90.000 deg
};
P[3034]{
   GP1:
	UF : 0, UT : 6,		CONFIG : 'N U T, 0, 0, 0',
	X =  485.554  mm,	Y =   -431.183  mm,	Z =   -251.124  mm,
	W =  90.000 deg,	P =   0.000 deg,	R =   90.000 deg
};
P[3035]{
   GP1:
	UF : 0, UT : 6,		CONFIG : 'N U T, 0, 0, 0',
	X =  486.742  mm,	Y =   -430.379  mm,	Z =   -251.410  mm,
	W =  90.000 deg,	P =   0.000 deg,	R =   90.000 deg
};
P[3036]{
   GP1:
	UF : 0, UT : 6,		CONFIG : 'N U T, 0, 0, 0',
	X =  489.127  mm,	Y =   -428.992  mm,	Z =   -251.434  mm,
	W =  90.000 deg,	P =   0.000 deg,	R =   90.000 deg
};
P[3037]{
   GP1:
	UF : 0, UT : 6,		CONFIG : 'N U T, 0, 0, 0',
	X =  490.843  mm,	Y =   -427.993  mm,	Z =   -251.453  mm,
	W =  90.000 deg,	P =   0.000 deg,	R =   90.000 deg
};
P[3038]{
   GP1:
	UF : 0, UT : 6,		CONFIG : 'N U T, 0, 0, 0',
	X =  491.774  mm,	Y =   -427.542  mm,	Z =   -251.244  mm,
	W =  90.000 deg,	P =   0.000 deg,	R =   90.000 deg
};
P[3039]{
   GP1:
	UF : 0, UT : 6,		CONFIG : 'N U T, 0, 0, 0',
	X =  493.019  mm,	Y =   -426.806  mm,	Z =   -251.288  mm,
	W =  90.000 deg,	P =   0.000 deg,	R =   90.000 deg
};
P[3040]{
   GP1:
	UF : 0, UT : 6,		CONFIG : 'N U T, 0, 0, 0',
	X =  494.155  mm,	Y =   -426.075  mm,	Z =   -251.470  mm,
	W =  90.000 deg,	P =   0.000 deg,	R =   90.000 deg
};
P[3041]{
   GP1:
	UF : 0, UT : 6,		CONFIG : 'N U T, 0, 0, 0',
	X =  495.329  mm,	Y =   -425.470  mm,	Z =   -251.290  mm,
	W =  90.000 deg,	P =   0.000 deg,	R =   90.000 deg
};
P[3042]{
   GP1:
	UF : 0, UT : 6,		CONFIG : 'N U T, 0, 0, 0',
	X =  496.759  mm,	Y =   -424.600  mm,	Z =   -251.401  mm,
	W =  90.000 deg,	P =   0.000 deg,	R =   90.000 deg
};
P[3043]{
   GP1:
	UF : 0, UT : 6,		CONFIG : 'N U T, 0, 0, 0',
	X =  498.263  mm,	Y =   -423.745  mm,	Z =   -251.367  mm,
	W =  90.000 deg,	P =   0.000 deg,	R =   90.000 deg
};
P[3044]{
   GP1:
	UF : 0, UT : 6,		CONFIG : 'N U T, 0, 0, 0',
	X =  503.030  mm,	Y =   -420.938  mm,	Z =   -251.499  mm,
	W =  90.000 deg,	P =   0.000 deg,	R =   90.000 deg
};
P[3045]{
   GP1:
	UF : 0, UT : 6,		CONFIG : 'N U T, 0, 0, 0',
	X =  504.449  mm,	Y =   -420.233  mm,	Z =   -251.222  mm,
	W =  90.000 deg,	P =   0.000 deg,	R =   90.000 deg
};
P[3046]{
   GP1:
	UF : 0, UT : 6,		CONFIG : 'N U T, 0, 0, 0',
	X =  507.671  mm,	Y =   -418.340  mm,	Z =   -251.301  mm,
	W =  90.000 deg,	P =   0.000 deg,	R =   90.000 deg
};
P[3047]{
   GP1:
	UF : 0, UT : 6,		CONFIG : 'N U T, 0, 0, 0',
	X =  508.421  mm,	Y =   -417.952  mm,	Z =   -251.191  mm,
	W =  90.000 deg,	P =   0.000 deg,	R =   90.000 deg
};
P[3048]{
   GP1:
	UF : 0, UT : 6,		CONFIG : 'N U T, 0, 0, 0',
	X =  509.227  mm,	Y =   -417.449  mm,	Z =   -251.282  mm,
	W =  90.000 deg,	P =   0.000 deg,	R =   90.000 deg
};
P[3049]{
   GP1:
	UF : 0, UT : 6,		CONFIG : 'N U T, 0, 0, 0',
	X =  512.965  mm,	Y =   -415.288  mm,	Z =   -251.289  mm,
	W =  90.000 deg,	P =   0.000 deg,	R =   90.000 deg
};
P[3050]{
   GP1:
	UF : 0, UT : 6,		CONFIG : 'N U T, 0, 0, 0',
	X =  514.505  mm,	Y =   -414.309  mm,	Z =   -251.508  mm,
	W =  90.000 deg,	P =   0.000 deg,	R =   90.000 deg
};
P[3051]{
   GP1:
	UF : 0, UT : 6,		CONFIG : 'N U T, 0, 0, 0',
	X =  515.860  mm,	Y =   -413.561  mm,	Z =   -251.425  mm,
	W =  90.000 deg,	P =   0.000 deg,	R =   90.000 deg
};
P[3052]{
   GP1:
	UF : 0, UT : 6,		CONFIG : 'N U T, 0, 0, 0',
	X =  516.842  mm,	Y =   -412.975  mm,	Z =   -251.468  mm,
	W =  90.000 deg,	P =   0.000 deg,	R =   90.000 deg
};
P[3053]{
   GP1:
	UF : 0, UT : 6,		CONFIG : 'N U T, 0, 0, 0',
	X =  519.969  mm,	Y =   -411.168  mm,	Z =   -251.475  mm,
	W =  90.000 deg,	P =   0.000 deg,	R =   90.000 deg
};
P[3054]{
   GP1:
	UF : 0, UT : 6,		CONFIG : 'N U T, 0, 0, 0',
	X =  521.150  mm,	Y =   -410.637  mm,	Z =   -251.106  mm,
	W =  90.000 deg,	P =   0.000 deg,	R =   90.000 deg
};
P[3055]{
   GP1:
	UF : 0, UT : 6,		CONFIG : 'N U T, 0, 0, 0',
	X =  523.861  mm,	Y =   -408.907  mm,	Z =   -251.506  mm,
	W =  90.000 deg,	P =   0.000 deg,	R =   90.000 deg
};
P[3056]{
   GP1:
	UF : 0, UT : 6,		CONFIG : 'N U T, 0, 0, 0',
	X =  525.496  mm,	Y =   -407.979  mm,	Z =   -251.467  mm,
	W =  90.000 deg,	P =   0.000 deg,	R =   90.000 deg
};
P[3057]{
   GP1:
	UF : 0, UT : 6,		CONFIG : 'N U T, 0, 0, 0',
	X =  526.372  mm,	Y =   -407.576  mm,	Z =   -251.218  mm,
	W =  90.000 deg,	P =   0.000 deg,	R =   90.000 deg
};
P[3058]{
   GP1:
	UF : 0, UT : 6,		CONFIG : 'N U T, 0, 0, 0',
	X =  528.212  mm,	Y =   -406.486  mm,	Z =   -251.287  mm,
	W =  90.000 deg,	P =   0.000 deg,	R =   90.000 deg
};
P[3059]{
   GP1:
	UF : 0, UT : 6,		CONFIG : 'N U T, 0, 0, 0',
	X =  530.453  mm,	Y =   -405.128  mm,	Z =   -251.441  mm,
	W =  90.000 deg,	P =   0.000 deg,	R =   90.000 deg
};
P[3060]{
   GP1:
	UF : 0, UT : 6,		CONFIG : 'N U T, 0, 0, 0',
	X =  531.631  mm,	Y =   -404.469  mm,	Z =   -251.389  mm,
	W =  90.000 deg,	P =   0.000 deg,	R =   90.000 deg
};
P[3061]{
   GP1:
	UF : 0, UT : 6,		CONFIG : 'N U T, 0, 0, 0',
	X =  533.209  mm,	Y =   -403.567  mm,	Z =   -251.367  mm,
	W =  90.000 deg,	P =   0.000 deg,	R =   90.000 deg
};
P[3062]{
   GP1:
	UF : 0, UT : 6,		CONFIG : 'N U T, 0, 0, 0',
	X =  534.147  mm,	Y =   -403.019  mm,	Z =   -251.382  mm,
	W =  90.000 deg,	P =   0.000 deg,	R =   90.000 deg
};
P[3063]{
   GP1:
	UF : 0, UT : 6,		CONFIG : 'N U T, 0, 0, 0',
	X =  535.717  mm,	Y =   -402.060  mm,	Z =   -251.510  mm,
	W =  90.000 deg,	P =   0.000 deg,	R =   90.000 deg
};
P[3064]{
   GP1:
	UF : 0, UT : 6,		CONFIG : 'N U T, 0, 0, 0',
	X =  537.605  mm,	Y =   -400.992  mm,	Z =   -251.373  mm,
	W =  90.000 deg,	P =   0.000 deg,	R =   90.000 deg
};
P[3065]{
   GP1:
	UF : 0, UT : 6,		CONFIG : 'N U T, 0, 0, 0',
	X =  538.669  mm,	Y =   -400.352  mm,	Z =   -251.133  mm,
	W =  90.000 deg,	P =   0.000 deg,	R =   90.000 deg
};
P[3066]{
   GP1:
	UF : 0, UT : 6,		CONFIG : 'N U T, 0, 0, 0',
	X =  541.356  mm,	Y =   -397.681  mm,	Z =   -251.457  mm,
	W =  90.000 deg,	P =   0.000 deg,	R =   90.000 deg
};
P[3067]{
   GP1:
	UF : 0, UT : 6,		CONFIG : 'N U T, 0, 0, 0',
	X =  542.359  mm,	Y =   -396.504  mm,	Z =   -251.110  mm,
	W =  90.000 deg,	P =   0.000 deg,	R =   90.000 deg
};
P[3068]{
   GP1:
	UF : 0, UT : 6,		CONFIG : 'N U T, 0, 0, 0',
	X =  544.419  mm,	Y =   -390.700  mm,	Z =   -251.051  mm,
	W =  90.000 deg,	P =   0.000 deg,	R =   90.000 deg
};
P[3069]{
   GP1:
	UF : 0, UT : 6,		CONFIG : 'N U T, 0, 0, 0',
	X =  544.210  mm,	Y =   -387.774  mm,	Z =   -251.424  mm,
	W =  90.000 deg,	P =   0.000 deg,	R =   90.000 deg
};
P[3070]{
   GP1:
	UF : 0, UT : 6,		CONFIG : 'N U T, 0, 0, 0',
	X =  544.219  mm,	Y =   -386.939  mm,	Z =   -251.077  mm,
	W =  90.000 deg,	P =   0.000 deg,	R =   90.000 deg
};
P[3071]{
   GP1:
	UF : 0, UT : 6,		CONFIG : 'N U T, 0, 0, 0',
	X =  543.614  mm,	Y =   -385.021  mm,	Z =   -251.373  mm,
	W =  90.000 deg,	P =   0.000 deg,	R =   90.000 deg
};
P[3072]{
   GP1:
	UF : 0, UT : 6,		CONFIG : 'N U T, 0, 0, 0',
	X =  542.654  mm,	Y =   -382.928  mm,	Z =   -251.446  mm,
	W =  90.000 deg,	P =   0.000 deg,	R =   90.000 deg
};
P[3073]{
   GP1:
	UF : 0, UT : 6,		CONFIG : 'N U T, 0, 0, 0',
	X =  542.292  mm,	Y =   -382.200  mm,	Z =   -251.477  mm,
	W =  90.000 deg,	P =   0.000 deg,	R =   90.000 deg
};
P[3074]{
   GP1:
	UF : 0, UT : 6,		CONFIG : 'N U T, 0, 0, 0',
	X =  541.377  mm,	Y =   -380.574  mm,	Z =   -251.429  mm,
	W =  90.000 deg,	P =   0.000 deg,	R =   90.000 deg
};
P[3075]{
   GP1:
	UF : 0, UT : 6,		CONFIG : 'N U T, 0, 0, 0',
	X =  540.542  mm,	Y =   -379.103  mm,	Z =   -251.395  mm,
	W =  90.000 deg,	P =   0.000 deg,	R =   90.000 deg
};
P[3076]{
   GP1:
	UF : 0, UT : 6,		CONFIG : 'N U T, 0, 0, 0',
	X =  539.905  mm,	Y =   -377.881  mm,	Z =   -251.228  mm,
	W =  90.000 deg,	P =   0.000 deg,	R =   90.000 deg
};
P[3077]{
   GP1:
	UF : 0, UT : 6,		CONFIG : 'N U T, 0, 0, 0',
	X =  538.657  mm,	Y =   -375.911  mm,	Z =   -251.496  mm,
	W =  90.000 deg,	P =   0.000 deg,	R =   90.000 deg
};
P[3078]{
   GP1:
	UF : 0, UT : 6,		CONFIG : 'N U T, 0, 0, 0',
	X =  537.641  mm,	Y =   -374.147  mm,	Z =   -251.489  mm,
	W =  90.000 deg,	P =   0.000 deg,	R =   90.000 deg
};
P[3079]{
   GP1:
	UF : 0, UT : 6,		CONFIG : 'N U T, 0, 0, 0',
	X =  537.289  mm,	Y =   -373.340  mm,	Z =   -251.214  mm,
	W =  90.000 deg,	P =   0.000 deg,	R =   90.000 deg
};
P[3080]{
   GP1:
	UF : 0, UT : 6,		CONFIG : 'N U T, 0, 0, 0',
	X =  536.597  mm,	Y =   -372.331  mm,	Z =   -251.478  mm,
	W =  90.000 deg,	P =   0.000 deg,	R =   90.000 deg
};
P[3081]{
   GP1:
	UF : 0, UT : 6,		CONFIG : 'N U T, 0, 0, 0',
	X =  536.015  mm,	Y =   -371.291  mm,	Z =   -251.434  mm,
	W =  90.000 deg,	P =   0.000 deg,	R =   90.000 deg
};
P[3082]{
   GP1:
	UF : 0, UT : 6,		CONFIG : 'N U T, 0, 0, 0',
	X =  535.632  mm,	Y =   -370.382  mm,	Z =   -251.090  mm,
	W =  90.000 deg,	P =   0.000 deg,	R =   90.000 deg
};
P[3083]{
   GP1:
	UF : 0, UT : 6,		CONFIG : 'N U T, 0, 0, 0',
	X =  534.528  mm,	Y =   -368.674  mm,	Z =   -251.375  mm,
	W =  90.000 deg,	P =   0.000 deg,	R =   90.000 deg
};
P[3084]{
   GP1:
	UF : 0, UT : 6,		CONFIG : 'N U T, 0, 0, 0',
	X =  533.991  mm,	Y =   -367.654  mm,	Z =   -251.248  mm,
	W =  90.000 deg,	P =   0.000 deg,	R =   90.000 deg
};
P[3085]{
   GP1:
	UF : 0, UT : 6,		CONFIG : 'N U T, 0, 0, 0',
	X =  533.554  mm,	Y =   -367.039  mm,	Z =   -251.450  mm,
	W =  90.000 deg,	P =   0.000 deg,	R =   90.000 deg
};
P[3086]{
   GP1:
	UF : 0, UT : 6,		CONFIG : 'N U T, 0, 0, 0',
	X =  533.281  mm,	Y =   -366.278  mm,	Z =   -251.043  mm,
	W =  90.000 deg,	P =   0.000 deg,	R =   90.000 deg
};
P[3087]{
   GP1:
	UF : 0, UT : 6,		CONFIG : 'N U T, 0, 0, 0',
	X =  532.576  mm,	Y =   -365.372  mm,	Z =   -251.485  mm,
	W =  90.000 deg,	P =   0.000 deg,	R =   90.000 deg
};
P[3088]{
   GP1:
	UF : 0, UT : 6,		CONFIG : 'N U T, 0, 0, 0',
	X =  532.156  mm,	Y =   -364.342  mm,	Z =   -251.064  mm,
	W =  90.000 deg,	P =   0.000 deg,	R =   90.000 deg
};
P[3089]{
   GP1:
	UF : 0, UT : 6,		CONFIG : 'N U T, 0, 0, 0',
	X =  531.140  mm,	Y =   -362.832  mm,	Z =   -251.413  mm,
	W =  90.000 deg,	P =   0.000 deg,	R =   90.000 deg
};
P[3090]{
   GP1:
	UF : 0, UT : 6,		CONFIG : 'N U T, 0, 0, 0',
	X =  530.285  mm,	Y =   -361.147  mm,	Z =   -251.126  mm,
	W =  90.000 deg,	P =   0.000 deg,	R =   90.000 deg
};
P[3091]{
   GP1:
	UF : 0, UT : 6,		CONFIG : 'N U T, 0, 0, 0',
	X =  529.220  mm,	Y =   -359.340  mm,	Z =   -251.178  mm,
	W =  90.000 deg,	P =   0.000 deg,	R =   90.000 deg
};
P[3092]{
   GP1:
	UF : 0, UT : 6,		CONFIG : 'N U T, 0, 0, 0',
	X =  528.824  mm,	Y =   -358.765  mm,	Z =   -251.334  mm,
	W =  90.000 deg,	P =   0.000 deg,	R =   90.000 deg
};
P[3093]{
   GP1:
	UF : 0, UT : 6,		CONFIG : 'N U T, 0, 0, 0',
	X =  527.293  mm,	Y =   -356.222  mm,	Z =   -251.483  mm,
	W =  90.000 deg,	P =   0.000 deg,	R =   90.000 deg
};
P[3094]{
   GP1:
	UF : 0, UT : 6,		CONFIG : 'N U T, 0, 0, 0',
	X =  526.452  mm,	Y =   -354.757  mm,	Z =   -251.473  mm,
	W =  90.000 deg,	P =   0.000 deg,	R =   90.000 deg
};
P[3095]{
   GP1:
	UF : 0, UT : 6,		CONFIG : 'N U T, 0, 0, 0',
	X =  524.805  mm,	Y =   -351.908  mm,	Z =   -251.479  mm,
	W =  90.000 deg,	P =   0.000 deg,	R =   90.000 deg
};
P[3096]{
   GP1:
	UF : 0, UT : 6,		CONFIG : 'N U T, 0, 0, 0',
	X =  523.808  mm,	Y =   -349.934  mm,	Z =   -251.131  mm,
	W =  90.000 deg,	P =   0.000 deg,	R =   90.000 deg
};
P[3097]{
   GP1:
	UF : 0, UT : 6,		CONFIG : 'N U T, 0, 0, 0',
	X =  521.287  mm,	Y =   -345.723  mm,	Z =   -251.352  mm,
	W =  90.000 deg,	P =   0.000 deg,	R =   90.000 deg
};
P[3098]{
   GP1:
	UF : 0, UT : 6,		CONFIG : 'N U T, 0, 0, 0',
	X =  519.040  mm,	Y =   -341.934  mm,	Z =   -251.494  mm,
	W =  90.000 deg,	P =   0.000 deg,	R =   90.000 deg
};
P[3099]{
   GP1:
	UF : 0, UT : 6,		CONFIG : 'N U T, 0, 0, 0',
	X =  517.885  mm,	Y =   -339.840  mm,	Z =   -251.360  mm,
	W =  90.000 deg,	P =   0.000 deg,	R =   90.000 deg
};
P[3100]{
   GP1:
	UF : 0, UT : 6,		CONFIG : 'N U T, 0, 0, 0',
	X =  517.062  mm,	Y =   -338.465  mm,	Z =   -251.432  mm,
	W =  90.000 deg,	P =   0.000 deg,	R =   90.000 deg
};
P[3101]{
   GP1:
	UF : 0, UT : 6,		CONFIG : 'N U T, 0, 0, 0',
	X =  516.343  mm,	Y =   -337.194  mm,	Z =   -251.397  mm,
	W =  90.000 deg,	P =   0.000 deg,	R =   90.000 deg
};
P[3102]{
   GP1:
	UF : 0, UT : 6,		CONFIG : 'N U T, 0, 0, 0',
	X =  515.785  mm,	Y =   -336.305  mm,	Z =   -251.503  mm,
	W =  90.000 deg,	P =   0.000 deg,	R =   90.000 deg
};
P[3103]{
   GP1:
	UF : 0, UT : 6,		CONFIG : 'N U T, 0, 0, 0',
	X =  513.732  mm,	Y =   -332.699  mm,	Z =   -251.434  mm,
	W =  90.000 deg,	P =   0.000 deg,	R =   90.000 deg
};
P[3104]{
   GP1:
	UF : 0, UT : 6,		CONFIG : 'N U T, 0, 0, 0',
	X =  513.231  mm,	Y =   -331.885  mm,	Z =   -251.510  mm,
	W =  90.000 deg,	P =   0.000 deg,	R =   90.000 deg
};
P[3105]{
   GP1:
	UF : 0, UT : 6,		CONFIG : 'N U T, 0, 0, 0',
	X =  512.651  mm,	Y =   -330.620  mm,	Z =   -251.146  mm,
	W =  90.000 deg,	P =   0.000 deg,	R =   90.000 deg
};
P[3106]{
   GP1:
	UF : 0, UT : 6,		CONFIG : 'N U T, 0, 0, 0',
	X =  511.522  mm,	Y =   -328.886  mm,	Z =   -251.455  mm,
	W =  90.000 deg,	P =   0.000 deg,	R =   90.000 deg
};
P[3107]{
   GP1:
	UF : 0, UT : 6,		CONFIG : 'N U T, 0, 0, 0',
	X =  506.835  mm,	Y =   -320.669  mm,	Z =   -251.314  mm,
	W =  90.000 deg,	P =   0.000 deg,	R =   90.000 deg
};
P[3108]{
   GP1:
	UF : 0, UT : 6,		CONFIG : 'N U T, 0, 0, 0',
	X =  504.012  mm,	Y =   -315.676  mm,	Z =   -251.171  mm,
	W =  90.000 deg,	P =   0.000 deg,	R =   90.000 deg
};
P[3109]{
   GP1:
	UF : 0, UT : 6,		CONFIG : 'N U T, 0, 0, 0',
	X =  502.975  mm,	Y =   -313.842  mm,	Z =   -251.117  mm,
	W =  90.000 deg,	P =   0.000 deg,	R =   90.000 deg
};
P[3110]{
   GP1:
	UF : 0, UT : 6,		CONFIG : 'N U T, 0, 0, 0',
	X =  501.058  mm,	Y =   -310.599  mm,	Z =   -251.225  mm,
	W =  90.000 deg,	P =   0.000 deg,	R =   90.000 deg
};
P[3111]{
   GP1:
	UF : 0, UT : 6,		CONFIG : 'N U T, 0, 0, 0',
	X =  500.417  mm,	Y =   -309.654  mm,	Z =   -251.457  mm,
	W =  90.000 deg,	P =   0.000 deg,	R =   90.000 deg
};
P[3112]{
   GP1:
	UF : 0, UT : 6,		CONFIG : 'N U T, 0, 0, 0',
	X =  500.151  mm,	Y =   -308.954  mm,	Z =   -251.119  mm,
	W =  90.000 deg,	P =   0.000 deg,	R =   90.000 deg
};
P[3113]{
   GP1:
	UF : 0, UT : 6,		CONFIG : 'N U T, 0, 0, 0',
	X =  499.586  mm,	Y =   -308.229  mm,	Z =   -251.477  mm,
	W =  90.000 deg,	P =   0.000 deg,	R =   90.000 deg
};
P[3114]{
   GP1:
	UF : 0, UT : 6,		CONFIG : 'N U T, 0, 0, 0',
	X =  498.516  mm,	Y =   -306.282  mm,	Z =   -251.345  mm,
	W =  90.000 deg,	P =   0.000 deg,	R =   90.000 deg
};
P[3115]{
   GP1:
	UF : 0, UT : 6,		CONFIG : 'N U T, 0, 0, 0',
	X =  496.833  mm,	Y =   -303.362  mm,	Z =   -251.338  mm,
	W =  90.000 deg,	P =   0.000 deg,	R =   90.000 deg
};
P[3116]{
   GP1:
	UF : 0, UT : 6,		CONFIG : 'N U T, 0, 0, 0',
	X =  496.007  mm,	Y =   -301.999  mm,	Z =   -251.431  mm,
	W =  90.000 deg,	P =   0.000 deg,	R =   90.000 deg
};
P[3117]{
   GP1:
	UF : 0, UT : 6,		CONFIG : 'N U T, 0, 0, 0',
	X =  495.500  mm,	Y =   -301.121  mm,	Z =   -251.432  mm,
	W =  90.000 deg,	P =   0.000 deg,	R =   90.000 deg
};
P[3118]{
   GP1:
	UF : 0, UT : 6,		CONFIG : 'N U T, 0, 0, 0',
	X =  493.047  mm,	Y =   -296.828  mm,	Z =   -251.368  mm,
	W =  90.000 deg,	P =   0.000 deg,	R =   90.000 deg
};
P[3119]{
   GP1:
	UF : 0, UT : 6,		CONFIG : 'N U T, 0, 0, 0',
	X =  492.096  mm,	Y =   -295.183  mm,	Z =   -251.374  mm,
	W =  90.000 deg,	P =   0.000 deg,	R =   90.000 deg
};
P[3120]{
   GP1:
	UF : 0, UT : 6,		CONFIG : 'N U T, 0, 0, 0',
	X =  491.551  mm,	Y =   -294.315  mm,	Z =   -251.480  mm,
	W =  90.000 deg,	P =   0.000 deg,	R =   90.000 deg
};
P[3121]{
   GP1:
	UF : 0, UT : 6,		CONFIG : 'N U T, 0, 0, 0',
	X =  490.912  mm,	Y =   -293.159  mm,	Z =   -251.411  mm,
	W =  90.000 deg,	P =   0.000 deg,	R =   90.000 deg
};
P[3122]{
   GP1:
	UF : 0, UT : 6,		CONFIG : 'N U T, 0, 0, 0',
	X =  490.126  mm,	Y =   -291.776  mm,	Z =   -251.380  mm,
	W =  90.000 deg,	P =   0.000 deg,	R =   90.000 deg
};
P[3123]{
   GP1:
	UF : 0, UT : 6,		CONFIG : 'N U T, 0, 0, 0',
	X =  489.521  mm,	Y =   -290.697  mm,	Z =   -251.335  mm,
	W =  90.000 deg,	P =   0.000 deg,	R =   90.000 deg
};
P[3124]{
   GP1:
	UF : 0, UT : 6,		CONFIG : 'N U T, 0, 0, 0',
	X =  489.032  mm,	Y =   -289.909  mm,	Z =   -251.418  mm,
	W =  90.000 deg,	P =   0.000 deg,	R =   90.000 deg
};
P[3125]{
   GP1:
	UF : 0, UT : 6,		CONFIG : 'N U T, 0, 0, 0',
	X =  488.626  mm,	Y =   -288.924  mm,	Z =   -251.026  mm,
	W =  90.000 deg,	P =   0.000 deg,	R =   90.000 deg
};
P[3126]{
   GP1:
	UF : 0, UT : 6,		CONFIG : 'N U T, 0, 0, 0',
	X =  487.655  mm,	Y =   -287.587  mm,	Z =   -251.506  mm,
	W =  90.000 deg,	P =   0.000 deg,	R =   90.000 deg
};
P[3127]{
   GP1:
	UF : 0, UT : 6,		CONFIG : 'N U T, 0, 0, 0',
	X =  486.801  mm,	Y =   -285.902  mm,	Z =   -251.219  mm,
	W =  90.000 deg,	P =   0.000 deg,	R =   90.000 deg
};
P[3128]{
   GP1:
	UF : 0, UT : 6,		CONFIG : 'N U T, 0, 0, 0',
	X =  485.515  mm,	Y =   -283.794  mm,	Z =   -251.384  mm,
	W =  90.000 deg,	P =   0.000 deg,	R =   90.000 deg
};
P[3129]{
   GP1:
	UF : 0, UT : 6,		CONFIG : 'N U T, 0, 0, 0',
	X =  485.179  mm,	Y =   -283.103  mm,	Z =   -251.231  mm,
	W =  90.000 deg,	P =   0.000 deg,	R =   90.000 deg
};
P[3130]{
   GP1:
	UF : 0, UT : 6,		CONFIG : 'N U T, 0, 0, 0',
	X =  483.547  mm,	Y =   -280.184  mm,	Z =   -251.104  mm,
	W =  90.000 deg,	P =   0.000 deg,	R =   90.000 deg
};
P[3131]{
   GP1:
	UF : 0, UT : 6,		CONFIG : 'N U T, 0, 0, 0',
	X =  482.442  mm,	Y =   -278.499  mm,	Z =   -251.421  mm,
	W =  90.000 deg,	P =   0.000 deg,	R =   90.000 deg
};
P[3132]{
   GP1:
	UF : 0, UT : 6,		CONFIG : 'N U T, 0, 0, 0',
	X =  481.902  mm,	Y =   -277.524  mm,	Z =   -251.366  mm,
	W =  90.000 deg,	P =   0.000 deg,	R =   90.000 deg
};
P[3133]{
   GP1:
	UF : 0, UT : 6,		CONFIG : 'N U T, 0, 0, 0',
	X =  480.724  mm,	Y =   -275.259  mm,	Z =   -251.051  mm,
	W =  90.000 deg,	P =   0.000 deg,	R =   90.000 deg
};
P[3134]{
   GP1:
	UF : 0, UT : 6,		CONFIG : 'N U T, 0, 0, 0',
	X =  477.455  mm,	Y =   -269.923  mm,	Z =   -251.509  mm,
	W =  90.000 deg,	P =   0.000 deg,	R =   90.000 deg
};
P[3135]{
   GP1:
	UF : 0, UT : 6,		CONFIG : 'N U T, 0, 0, 0',
	X =  476.117  mm,	Y =   -267.322  mm,	Z =   -251.112  mm,
	W =  90.000 deg,	P =   0.000 deg,	R =   90.000 deg
};
P[3136]{
   GP1:
	UF : 0, UT : 6,		CONFIG : 'N U T, 0, 0, 0',
	X =  474.550  mm,	Y =   -264.871  mm,	Z =   -251.479  mm,
	W =  90.000 deg,	P =   0.000 deg,	R =   90.000 deg
};
P[3137]{
   GP1:
	UF : 0, UT : 6,		CONFIG : 'N U T, 0, 0, 0',
	X =  473.498  mm,	Y =   -262.980  mm,	Z =   -251.382  mm,
	W =  90.000 deg,	P =   0.000 deg,	R =   90.000 deg
};
P[3138]{
   GP1:
	UF : 0, UT : 6,		CONFIG : 'N U T, 0, 0, 0',
	X =  472.872  mm,	Y =   -261.943  mm,	Z =   -251.448  mm,
	W =  90.000 deg,	P =   0.000 deg,	R =   90.000 deg
};
P[3139]{
   GP1:
	UF : 0, UT : 6,		CONFIG : 'N U T, 0, 0, 0',
	X =  471.547  mm,	Y =   -259.555  mm,	Z =   -251.320  mm,
	W =  90.000 deg,	P =   0.000 deg,	R =   90.000 deg
};
P[3140]{
   GP1:
	UF : 0, UT : 6,		CONFIG : 'N U T, 0, 0, 0',
	X =  469.677  mm,	Y =   -256.318  mm,	Z =   -251.320  mm,
	W =  90.000 deg,	P =   0.000 deg,	R =   90.000 deg
};
P[3141]{
   GP1:
	UF : 0, UT : 6,		CONFIG : 'N U T, 0, 0, 0',
	X =  469.234  mm,	Y =   -255.583  mm,	Z =   -251.368  mm,
	W =  90.000 deg,	P =   0.000 deg,	R =   90.000 deg
};
P[3142]{
   GP1:
	UF : 0, UT : 6,		CONFIG : 'N U T, 0, 0, 0',
	X =  467.237  mm,	Y =   -252.074  mm,	Z =   -251.297  mm,
	W =  90.000 deg,	P =   0.000 deg,	R =   90.000 deg
};
P[3143]{
   GP1:
	UF : 0, UT : 6,		CONFIG : 'N U T, 0, 0, 0',
	X =  466.350  mm,	Y =   -250.562  mm,	Z =   -251.328  mm,
	W =  90.000 deg,	P =   0.000 deg,	R =   90.000 deg
};
P[3144]{
   GP1:
	UF : 0, UT : 6,		CONFIG : 'N U T, 0, 0, 0',
	X =  464.706  mm,	Y =   -247.695  mm,	Z =   -251.301  mm,
	W =  90.000 deg,	P =   0.000 deg,	R =   90.000 deg
};
P[3145]{
   GP1:
	UF : 0, UT : 6,		CONFIG : 'N U T, 0, 0, 0',
	X =  462.101  mm,	Y =   -243.322  mm,	Z =   -251.495  mm,
	W =  90.000 deg,	P =   0.000 deg,	R =   90.000 deg
};
P[3146]{
   GP1:
	UF : 0, UT : 6,		CONFIG : 'N U T, 0, 0, 0',
	X =  461.653  mm,	Y =   -242.554  mm,	Z =   -251.506  mm,
	W =  90.000 deg,	P =   0.000 deg,	R =   90.000 deg
};
P[3147]{
   GP1:
	UF : 0, UT : 6,		CONFIG : 'N U T, 0, 0, 0',
	X =  460.289  mm,	Y =   -240.164  mm,	Z =   -251.467  mm,
	W =  90.000 deg,	P =   0.000 deg,	R =   90.000 deg
};
P[3148]{
   GP1:
	UF : 0, UT : 6,		CONFIG : 'N U T, 0, 0, 0',
	X =  459.773  mm,	Y =   -239.241  mm,	Z =   -251.427  mm,
	W =  90.000 deg,	P =   0.000 deg,	R =   90.000 deg
};
P[3149]{
   GP1:
	UF : 0, UT : 6,		CONFIG : 'N U T, 0, 0, 0',
	X =  458.371  mm,	Y =   -236.687  mm,	Z =   -251.253  mm,
	W =  90.000 deg,	P =   0.000 deg,	R =   90.000 deg
};
P[3150]{
   GP1:
	UF : 0, UT : 6,		CONFIG : 'N U T, 0, 0, 0',
	X =  455.822  mm,	Y =   -232.250  mm,	Z =   -251.219  mm,
	W =  90.000 deg,	P =   0.000 deg,	R =   90.000 deg
};
P[3151]{
   GP1:
	UF : 0, UT : 6,		CONFIG : 'N U T, 0, 0, 0',
	X =  454.549  mm,	Y =   -230.240  mm,	Z =   -251.494  mm,
	W =  90.000 deg,	P =   0.000 deg,	R =   90.000 deg
};
P[3152]{
   GP1:
	UF : 0, UT : 6,		CONFIG : 'N U T, 0, 0, 0',
	X =  452.253  mm,	Y =   -226.131  mm,	Z =   -251.308  mm,
	W =  90.000 deg,	P =   0.000 deg,	R =   90.000 deg
};
P[3153]{
   GP1:
	UF : 0, UT : 6,		CONFIG : 'N U T, 0, 0, 0',
	X =  451.047  mm,	Y =   -223.958  mm,	Z =   -251.188  mm,
	W =  90.000 deg,	P =   0.000 deg,	R =   90.000 deg
};
P[3154]{
   GP1:
	UF : 0, UT : 6,		CONFIG : 'N U T, 0, 0, 0',
	X =  450.366  mm,	Y =   -222.755  mm,	Z =   -251.157  mm,
	W =  90.000 deg,	P =   0.000 deg,	R =   90.000 deg
};
P[3155]{
   GP1:
	UF : 0, UT : 6,		CONFIG : 'N U T, 0, 0, 0',
	X =  449.391  mm,	Y =   -221.258  mm,	Z =   -251.425  mm,
	W =  90.000 deg,	P =   0.000 deg,	R =   90.000 deg
};
P[3156]{
   GP1:
	UF : 0, UT : 6,		CONFIG : 'N U T, 0, 0, 0',
	X =  448.785  mm,	Y =   -220.204  mm,	Z =   -251.417  mm,
	W =  90.000 deg,	P =   0.000 deg,	R =   90.000 deg
};
P[3157]{
   GP1:
	UF : 0, UT : 6,		CONFIG : 'N U T, 0, 0, 0',
	X =  447.682  mm,	Y =   -218.326  mm,	Z =   -251.462  mm,
	W =  90.000 deg,	P =   0.000 deg,	R =   90.000 deg
};
P[3158]{
   GP1:
	UF : 0, UT : 6,		CONFIG : 'N U T, 0, 0, 0',
	X =  447.135  mm,	Y =   -217.408  mm,	Z =   -251.505  mm,
	W =  90.000 deg,	P =   0.000 deg,	R =   90.000 deg
};
P[3159]{
   GP1:
	UF : 0, UT : 6,		CONFIG : 'N U T, 0, 0, 0',
	X =  445.337  mm,	Y =   -214.170  mm,	Z =   -251.332  mm,
	W =  90.000 deg,	P =   0.000 deg,	R =   90.000 deg
};
P[3160]{
   GP1:
	UF : 0, UT : 6,		CONFIG : 'N U T, 0, 0, 0',
	X =  444.769  mm,	Y =   -213.131  mm,	Z =   -251.254  mm,
	W =  90.000 deg,	P =   0.000 deg,	R =   90.000 deg
};
P[3161]{
   GP1:
	UF : 0, UT : 6,		CONFIG : 'N U T, 0, 0, 0',
	X =  444.348  mm,	Y =   -212.471  mm,	Z =   -251.352  mm,
	W =  90.000 deg,	P =   0.000 deg,	R =   90.000 deg
};
P[3162]{
   GP1:
	UF : 0, UT : 6,		CONFIG : 'N U T, 0, 0, 0',
	X =  443.890  mm,	Y =   -211.615  mm,	Z =   -251.264  mm,
	W =  90.000 deg,	P =   0.000 deg,	R =   90.000 deg
};
P[3163]{
   GP1:
	UF : 0, UT : 6,		CONFIG : 'N U T, 0, 0, 0',
	X =  441.636  mm,	Y =   -207.550  mm,	Z =   -251.037  mm,
	W =  90.000 deg,	P =   0.000 deg,	R =   90.000 deg
};
P[3164]{
   GP1:
	UF : 0, UT : 6,		CONFIG : 'N U T, 0, 0, 0',
	X =  441.038  mm,	Y =   -206.779  mm,	Z =   -251.408  mm,
	W =  90.000 deg,	P =   0.000 deg,	R =   90.000 deg
};
P[3165]{
   GP1:
	UF : 0, UT : 6,		CONFIG : 'N U T, 0, 0, 0',
	X =  440.607  mm,	Y =   -205.797  mm,	Z =   -251.076  mm,
	W =  90.000 deg,	P =   0.000 deg,	R =   90.000 deg
};
P[3166]{
   GP1:
	UF : 0, UT : 6,		CONFIG : 'N U T, 0, 0, 0',
	X =  439.035  mm,	Y =   -203.243  mm,	Z =   -251.313  mm,
	W =  90.000 deg,	P =   0.000 deg,	R =   90.000 deg
};
P[3167]{
   GP1:
	UF : 0, UT : 6,		CONFIG : 'N U T, 0, 0, 0',
	X =  438.311  mm,	Y =   -202.117  mm,	Z =   -251.494  mm,
	W =  90.000 deg,	P =   0.000 deg,	R =   90.000 deg
};
P[3168]{
   GP1:
	UF : 0, UT : 6,		CONFIG : 'N U T, 0, 0, 0',
	X =  437.742  mm,	Y =   -201.079  mm,	Z =   -251.420  mm,
	W =  90.000 deg,	P =   0.000 deg,	R =   90.000 deg
};
P[3169]{
   GP1:
	UF : 0, UT : 6,		CONFIG : 'N U T, 0, 0, 0',
	X =  437.185  mm,	Y =   -200.164  mm,	Z =   -251.487  mm,
	W =  90.000 deg,	P =   0.000 deg,	R =   90.000 deg
};
P[3170]{
   GP1:
	UF : 0, UT : 6,		CONFIG : 'N U T, 0, 0, 0',
	X =  436.846  mm,	Y =   -199.239  mm,	Z =   -251.017  mm,
	W =  90.000 deg,	P =   0.000 deg,	R =   90.000 deg
};
P[3171]{
   GP1:
	UF : 0, UT : 6,		CONFIG : 'N U T, 0, 0, 0',
	X =  436.354  mm,	Y =   -198.685  mm,	Z =   -251.432  mm,
	W =  90.000 deg,	P =   0.000 deg,	R =   90.000 deg
};
P[3172]{
   GP1:
	UF : 0, UT : 6,		CONFIG : 'N U T, 0, 0, 0',
	X =  435.263  mm,	Y =   -196.706  mm,	Z =   -251.309  mm,
	W =  90.000 deg,	P =   0.000 deg,	R =   90.000 deg
};
P[3173]{
   GP1:
	UF : 0, UT : 6,		CONFIG : 'N U T, 0, 0, 0',
	X =  434.547  mm,	Y =   -195.374  mm,	Z =   -251.177  mm,
	W =  90.000 deg,	P =   0.000 deg,	R =   90.000 deg
};
P[3174]{
   GP1:
	UF : 0, UT : 6,		CONFIG : 'N U T, 0, 0, 0',
	X =  433.540  mm,	Y =   -193.547  mm,	Z =   -251.062  mm,
	W =  90.000 deg,	P =   0.000 deg,	R =   90.000 deg
};
P[3175]{
   GP1:
	UF : 0, UT : 6,		CONFIG : 'N U T, 0, 0, 0',
	X =  432.729  mm,	Y =   -192.381  mm,	Z =   -251.397  mm,
	W =  90.000 deg,	P =   0.000 deg,	R =   90.000 deg
};
P[3176]{
   GP1:
	UF : 0, UT : 6,		CONFIG : 'N U T, 0, 0, 0',
	X =  432.237  mm,	Y =   -191.307  mm,	Z =   -251.087  mm,
	W =  90.000 deg,	P =   0.000 deg,	R =   90.000 deg
};
P[3177]{
   GP1:
	UF : 0, UT : 6,		CONFIG : 'N U T, 0, 0, 0',
	X =  431.602  mm,	Y =   -190.198  mm,	Z =   -251.074  mm,
	W =  90.000 deg,	P =   0.000 deg,	R =   90.000 deg
};
P[3178]{
   GP1:
	UF : 0, UT : 6,		CONFIG : 'N U T, 0, 0, 0',
	X =  431.038  mm,	Y =   -189.516  mm,	Z =   -251.487  mm,
	W =  90.000 deg,	P =   0.000 deg,	R =   90.000 deg
};
P[3179]{
   GP1:
	UF : 0, UT : 6,		CONFIG : 'N U T, 0, 0, 0',
	X =  428.995  mm,	Y =   -185.945  mm,	Z =   -251.440  mm,
	W =  90.000 deg,	P =   0.000 deg,	R =   90.000 deg
};
P[3180]{
   GP1:
	UF : 0, UT : 6,		CONFIG : 'N U T, 0, 0, 0',
	X =  428.625  mm,	Y =   -185.345  mm,	Z =   -251.498  mm,
	W =  90.000 deg,	P =   0.000 deg,	R =   90.000 deg
};
P[3181]{
   GP1:
	UF : 0, UT : 6,		CONFIG : 'N U T, 0, 0, 0',
	X =  426.729  mm,	Y =   -181.911  mm,	Z =   -251.287  mm,
	W =  90.000 deg,	P =   0.000 deg,	R =   90.000 deg
};
P[3182]{
   GP1:
	UF : 0, UT : 6,		CONFIG : 'N U T, 0, 0, 0',
	X =  426.113  mm,	Y =   -180.668  mm,	Z =   -251.041  mm,
	W =  90.000 deg,	P =   0.000 deg,	R =   90.000 deg
};
P[3183]{
   GP1:
	UF : 0, UT : 6,		CONFIG : 'N U T, 0, 0, 0',
	X =  425.660  mm,	Y =   -179.893  mm,	Z =   -251.055  mm,
	W =  90.000 deg,	P =   0.000 deg,	R =   90.000 deg
};
P[3184]{
   GP1:
	UF : 0, UT : 6,		CONFIG : 'N U T, 0, 0, 0',
	X =  425.172  mm,	Y =   -179.352  mm,	Z =   -251.479  mm,
	W =  90.000 deg,	P =   0.000 deg,	R =   90.000 deg
};
P[3185]{
   GP1:
	UF : 0, UT : 6,		CONFIG : 'N U T, 0, 0, 0',
	X =  424.070  mm,	Y =   -177.287  mm,	Z =   -251.260  mm,
	W =  90.000 deg,	P =   0.000 deg,	R =   90.000 deg
};
P[3186]{
   GP1:
	UF : 0, UT : 6,		CONFIG : 'N U T, 0, 0, 0',
	X =  420.949  mm,	Y =   -172.005  mm,	Z =   -251.432  mm,
	W =  90.000 deg,	P =   0.000 deg,	R =   90.000 deg
};
P[3187]{
   GP1:
	UF : 0, UT : 6,		CONFIG : 'N U T, 0, 0, 0',
	X =  418.776  mm,	Y =   -168.175  mm,	Z =   -251.339  mm,
	W =  90.000 deg,	P =   0.000 deg,	R =   90.000 deg
};
P[3188]{
   GP1:
	UF : 0, UT : 6,		CONFIG : 'N U T, 0, 0, 0',
	X =  417.283  mm,	Y =   -165.497  mm,	Z =   -251.211  mm,
	W =  90.000 deg,	P =   0.000 deg,	R =   90.000 deg
};
P[3189]{
   GP1:
	UF : 0, UT : 6,		CONFIG : 'N U T, 0, 0, 0',
	X =  416.755  mm,	Y =   -164.688  mm,	Z =   -251.359  mm,
	W =  90.000 deg,	P =   0.000 deg,	R =   90.000 deg
};
P[3190]{
   GP1:
	UF : 0, UT : 6,		CONFIG : 'N U T, 0, 0, 0',
	X =  416.172  mm,	Y =   -163.643  mm,	Z =   -251.311  mm,
	W =  90.000 deg,	P =   0.000 deg,	R =   90.000 deg
};
P[3191]{
   GP1:
	UF : 0, UT : 6,		CONFIG : 'N U T, 0, 0, 0',
	X =  415.173  mm,	Y =   -161.923  mm,	Z =   -251.324  mm,
	W =  90.000 deg,	P =   0.000 deg,	R =   90.000 deg
};
P[3192]{
   GP1:
	UF : 0, UT : 6,		CONFIG : 'N U T, 0, 0, 0',
	X =  414.182  mm,	Y =   -160.254  mm,	Z =   -251.388  mm,
	W =  90.000 deg,	P =   0.000 deg,	R =   90.000 deg
};
P[3193]{
   GP1:
	UF : 0, UT : 6,		CONFIG : 'N U T, 0, 0, 0',
	X =  413.400  mm,	Y =   -158.951  mm,	Z =   -251.462  mm,
	W =  90.000 deg,	P =   0.000 deg,	R =   90.000 deg
};
P[3194]{
   GP1:
	UF : 0, UT : 6,		CONFIG : 'N U T, 0, 0, 0',
	X =  412.319  mm,	Y =   -157.048  mm,	Z =   -251.420  mm,
	W =  90.000 deg,	P =   0.000 deg,	R =   90.000 deg
};
P[3195]{
   GP1:
	UF : 0, UT : 6,		CONFIG : 'N U T, 0, 0, 0',
	X =  411.424  mm,	Y =   -155.499  mm,	Z =   -251.421  mm,
	W =  90.000 deg,	P =   0.000 deg,	R =   90.000 deg
};
P[3196]{
   GP1:
	UF : 0, UT : 6,		CONFIG : 'N U T, 0, 0, 0',
	X =  410.868  mm,	Y =   -154.559  mm,	Z =   -251.452  mm,
	W =  90.000 deg,	P =   0.000 deg,	R =   90.000 deg
};
P[3197]{
   GP1:
	UF : 0, UT : 6,		CONFIG : 'N U T, 0, 0, 0',
	X =  409.876  mm,	Y =   -152.860  mm,	Z =   -251.479  mm,
	W =  90.000 deg,	P =   0.000 deg,	R =   90.000 deg
};
P[3198]{
   GP1:
	UF : 0, UT : 6,		CONFIG : 'N U T, 0, 0, 0',
	X =  409.097  mm,	Y =   -151.491  mm,	Z =   -251.452  mm,
	W =  90.000 deg,	P =   0.000 deg,	R =   90.000 deg
};
P[3199]{
   GP1:
	UF : 0, UT : 6,		CONFIG : 'N U T, 0, 0, 0',
	X =  408.502  mm,	Y =   -150.416  mm,	Z =   -251.390  mm,
	W =  90.000 deg,	P =   0.000 deg,	R =   90.000 deg
};
P[3200]{
   GP1:
	UF : 0, UT : 6,		CONFIG : 'N U T, 0, 0, 0',
	X =  407.903  mm,	Y =   -149.170  mm,	Z =   -251.098  mm,
	W =  90.000 deg,	P =   0.000 deg,	R =   90.000 deg
};
P[3201]{
   GP1:
	UF : 0, UT : 6,		CONFIG : 'N U T, 0, 0, 0',
	X =  406.649  mm,	Y =   -147.107  mm,	Z =   -251.249  mm,
	W =  90.000 deg,	P =   0.000 deg,	R =   90.000 deg
};
P[3202]{
   GP1:
	UF : 0, UT : 6,		CONFIG : 'N U T, 0, 0, 0',
	X =  405.355  mm,	Y =   -145.021  mm,	Z =   -251.466  mm,
	W =  90.000 deg,	P =   0.000 deg,	R =   90.000 deg
};
P[3203]{
   GP1:
	UF : 0, UT : 6,		CONFIG : 'N U T, 0, 0, 0',
	X =  402.951  mm,	Y =   -140.769  mm,	Z =   -251.341  mm,
	W =  90.000 deg,	P =   0.000 deg,	R =   90.000 deg
};
P[3204]{
   GP1:
	UF : 0, UT : 6,		CONFIG : 'N U T, 0, 0, 0',
	X =  400.398  mm,	Y =   -136.250  mm,	Z =   -251.206  mm,
	W =  90.000 deg,	P =   0.000 deg,	R =   90.000 deg
};
P[3205]{
   GP1:
	UF : 0, UT : 6,		CONFIG : 'N U T, 0, 0, 0',
	X =  398.021  mm,	Y =   -132.308  mm,	Z =   -251.452  mm,
	W =  90.000 deg,	P =   0.000 deg,	R =   90.000 deg
};
P[3206]{
   GP1:
	UF : 0, UT : 6,		CONFIG : 'N U T, 0, 0, 0',
	X =  396.764  mm,	Y =   -130.174  mm,	Z =   -251.511  mm,
	W =  90.000 deg,	P =   0.000 deg,	R =   90.000 deg
};
P[3207]{
   GP1:
	UF : 0, UT : 6,		CONFIG : 'N U T, 0, 0, 0',
	X =  395.817  mm,	Y =   -128.283  mm,	Z =   -251.162  mm,
	W =  90.000 deg,	P =   0.000 deg,	R =   90.000 deg
};
P[3208]{
   GP1:
	UF : 0, UT : 6,		CONFIG : 'N U T, 0, 0, 0',
	X =  395.351  mm,	Y =   -127.620  mm,	Z =   -251.361  mm,
	W =  90.000 deg,	P =   0.000 deg,	R =   90.000 deg
};
P[3209]{
   GP1:
	UF : 0, UT : 6,		CONFIG : 'N U T, 0, 0, 0',
	X =  394.247  mm,	Y =   -125.676  mm,	Z =   -251.316  mm,
	W =  90.000 deg,	P =   0.000 deg,	R =   90.000 deg
};
P[3210]{
   GP1:
	UF : 0, UT : 6,		CONFIG : 'N U T, 0, 0, 0',
	X =  393.744  mm,	Y =   -124.629  mm,	Z =   -251.071  mm,
	W =  90.000 deg,	P =   0.000 deg,	R =   90.000 deg
};
P[3211]{
   GP1:
	UF : 0, UT : 6,		CONFIG : 'N U T, 0, 0, 0',
	X =  391.743  mm,	Y =   -121.129  mm,	Z =   -251.020  mm,
	W =  90.000 deg,	P =   0.000 deg,	R =   90.000 deg
};
P[3212]{
   GP1:
	UF : 0, UT : 6,		CONFIG : 'N U T, 0, 0, 0',
	X =  390.969  mm,	Y =   -120.020  mm,	Z =   -251.347  mm,
	W =  90.000 deg,	P =   0.000 deg,	R =   90.000 deg
};
P[3213]{
   GP1:
	UF : 0, UT : 6,		CONFIG : 'N U T, 0, 0, 0',
	X =  390.333  mm,	Y =   -118.875  mm,	Z =   -251.286  mm,
	W =  90.000 deg,	P =   0.000 deg,	R =   90.000 deg
};
P[3214]{
   GP1:
	UF : 0, UT : 6,		CONFIG : 'N U T, 0, 0, 0',
	X =  389.357  mm,	Y =   -117.153  mm,	Z =   -251.242  mm,
	W =  90.000 deg,	P =   0.000 deg,	R =   90.000 deg
};
P[3215]{
   GP1:
	UF : 0, UT : 6,		CONFIG : 'N U T, 0, 0, 0',
	X =  387.698  mm,	Y =   -114.350  mm,	Z =   -251.339  mm,
	W =  90.000 deg,	P =   0.000 deg,	R =   90.000 deg
};
P[3216]{
   GP1:
	UF : 0, UT : 6,		CONFIG : 'N U T, 0, 0, 0',
	X =  383.549  mm,	Y =   -107.281  mm,	Z =   -251.503  mm,
	W =  90.000 deg,	P =   0.000 deg,	R =   90.000 deg
};
P[3217]{
   GP1:
	UF : 0, UT : 6,		CONFIG : 'N U T, 0, 0, 0',
	X =  382.899  mm,	Y =   -106.052  mm,	Z =   -251.359  mm,
	W =  90.000 deg,	P =   0.000 deg,	R =   90.000 deg
};
P[3218]{
   GP1:
	UF : 0, UT : 6,		CONFIG : 'N U T, 0, 0, 0',
	X =  382.592  mm,	Y =   -105.381  mm,	Z =   -251.163  mm,
	W =  90.000 deg,	P =   0.000 deg,	R =   90.000 deg
};
P[3219]{
   GP1:
	UF : 0, UT : 6,		CONFIG : 'N U T, 0, 0, 0',
	X =  381.850  mm,	Y =   -104.318  mm,	Z =   -251.475  mm,
	W =  90.000 deg,	P =   0.000 deg,	R =   90.000 deg
};
P[3220]{
   GP1:
	UF : 0, UT : 6,		CONFIG : 'N U T, 0, 0, 0',
	X =  380.974  mm,	Y =   -102.729  mm,	Z =   -251.376  mm,
	W =  90.000 deg,	P =   0.000 deg,	R =   90.000 deg
};
P[3221]{
   GP1:
	UF : 0, UT : 6,		CONFIG : 'N U T, 0, 0, 0',
	X =  378.425  mm,	Y =   -98.317  mm,	Z =   -251.380  mm,
	W =  90.000 deg,	P =   0.000 deg,	R =   90.000 deg
};
P[3222]{
   GP1:
	UF : 0, UT : 6,		CONFIG : 'N U T, 0, 0, 0',
	X =  377.686  mm,	Y =   -96.801  mm,	Z =   -251.048  mm,
	W =  90.000 deg,	P =   0.000 deg,	R =   90.000 deg
};
P[3223]{
   GP1:
	UF : 0, UT : 6,		CONFIG : 'N U T, 0, 0, 0',
	X =  376.274  mm,	Y =   -94.357  mm,	Z =   -251.049  mm,
	W =  90.000 deg,	P =   0.000 deg,	R =   90.000 deg
};
P[3224]{
   GP1:
	UF : 0, UT : 6,		CONFIG : 'N U T, 0, 0, 0',
	X =  375.867  mm,	Y =   -93.750  mm,	Z =   -251.185  mm,
	W =  90.000 deg,	P =   0.000 deg,	R =   90.000 deg
};
P[3225]{
   GP1:
	UF : 0, UT : 6,		CONFIG : 'N U T, 0, 0, 0',
	X =  374.775  mm,	Y =   -91.789  mm,	Z =   -251.086  mm,
	W =  90.000 deg,	P =   0.000 deg,	R =   90.000 deg
};
P[3226]{
   GP1:
	UF : 0, UT : 6,		CONFIG : 'N U T, 0, 0, 0',
	X =  373.196  mm,	Y =   -89.234  mm,	Z =   -251.341  mm,
	W =  90.000 deg,	P =   0.000 deg,	R =   90.000 deg
};
P[3227]{
   GP1:
	UF : 0, UT : 6,		CONFIG : 'N U T, 0, 0, 0',
	X =  372.493  mm,	Y =   -87.993  mm,	Z =   -251.306  mm,
	W =  90.000 deg,	P =   0.000 deg,	R =   90.000 deg
};
P[3228]{
   GP1:
	UF : 0, UT : 6,		CONFIG : 'N U T, 0, 0, 0',
	X =  371.675  mm,	Y =   -86.501  mm,	Z =   -251.203  mm,
	W =  90.000 deg,	P =   0.000 deg,	R =   90.000 deg
};
P[3229]{
   GP1:
	UF : 0, UT : 6,		CONFIG : 'N U T, 0, 0, 0',
	X =  369.180  mm,	Y =   -82.458  mm,	Z =   -251.282  mm,
	W =  90.000 deg,	P =   0.000 deg,	R =   90.000 deg
};
P[3230]{
   GP1:
	UF : 0, UT : 6,		CONFIG : 'N U T, 0, 0, 0',
	X =  368.504  mm,	Y =   -81.554  mm,	Z =   -251.351  mm,
	W =  90.000 deg,	P =   0.000 deg,	R =   90.000 deg
};
P[3231]{
   GP1:
	UF : 0, UT : 6,		CONFIG : 'N U T, 0, 0, 0',
	X =  367.989  mm,	Y =   -80.735  mm,	Z =   -251.027  mm,
	W =  90.000 deg,	P =   0.000 deg,	R =   90.000 deg
};
P[3232]{
   GP1:
	UF : 0, UT : 6,		CONFIG : 'N U T, 0, 0, 0',
	X =  367.209  mm,	Y =   -80.216  mm,	Z =   -251.403  mm,
	W =  90.000 deg,	P =   0.000 deg,	R =   90.000 deg
};
P[3233]{
   GP1:
	UF : 0, UT : 6,		CONFIG : 'N U T, 0, 0, 0',
	X =  366.615  mm,	Y =   -79.701  mm,	Z =   -251.484  mm,
	W =  90.000 deg,	P =   0.000 deg,	R =   90.000 deg
};
P[3234]{
   GP1:
	UF : 0, UT : 6,		CONFIG : 'N U T, 0, 0, 0',
